		  CASE uiBothStep OF
           		0://	
					BoxReady_1st := FALSE;
					BoxReady_2nd := FALSE;					
					uiBothStep:=1000;	
	
				1000:
						BoxReady_1st:=TRUE;
						uiBothStep:=2000;
						
				2000:
						IF Robot._DI1.Notification THEN
							uiBothStep:=3000;
						END_IF
				3000:
					
					
						uiBothStep:=9000;	
					
				9000:
						BoxReady_2nd:=TRUE;
						uiBothStep:=9999;
				
				9999: //Wait		
        // wait reset
        END_CASE

       	  // Robot Abs move
           		 Robot.M_StartRobotAbsMove( GetBox:=Get,
											UseClampA:=UseA,
											UseClampB:=UseB,
											Area:=Area,
											ClampA_Address:=Address_A,
											ClampB_Address:=Address_B,
											BoxReady_1:=BoxReady_1st,
											BoxReady_2:=BoxReady_2nd);	
		
		
        IF Robot._DI1.Done THEN
			tonTimeOut.IN:=FALSE;
            uiExecutingStep := 30080;
        END_IF
		IF tonTimeOut.Q=TRUE THEN
				tonTimeOut.IN:=FALSE;
				strStatus :='FB_ShippingRobot_Left Step 30000: Reset Robot timeout';
				_Error:=TRUE;
			END_IF
    30080: // Check robot command is clear
        
        Robot.M_ResetRobotAbsMove(UseA,UseB);

        IF NOT Robot._DI1.Done THEN
			tonTimeOut.IN:=FALSE;
            uiExecutingStep := 90000; // go to place step
        END_IF    
   		tonTimeOut.IN:=TRUE;
		IF tonTimeOut.Q=TRUE THEN
			strStatus :='FB_ShippingRobot_Left Step 30080: Stop Robot timeout';
			_Error:=TRUE;
		END_IF
		
	90000:
			IF bCompleteRequest THEN
				uiExecutingStep := 91000;
			ELSE
				uiExecutingStep := 99000;
			END_IF
			
	91000:	// shipping allocate mission complete signal
		BuzzBlinker(ENABLE:=TRUE , TIMELOW:=T#0.3S , TIMEHIGH:=T#0.3S , OUT=> Buzz);
		LightBlinker(ENABLE := TRUE , TIMELOW := T#0.3S , TIMEHIGH := T#0.3S , OUT => RedLamp );
		TrigBuzz(CLK:=Buzz);
		TrigLight(CLK :=RedLamp);
		IF TrigBuzz.Q THEN
			BlinkInfo.BuzzCount := BlinkInfo.BuzzCount +1;
		END_IF
		IF TrigLight.Q THEN
			BlinkInfo.LightCount := BlinkInfo.LightCount +1;
		END_IF
		
		IF BlinkInfo.BuzzCount >= BlinkInfo.MaxBuzzCOunt AND BlinkInfo.LightCount >=BlinkInfo.MaxLightCount THEN
			TON_BlinkDelay.IN :=TRUE;
			IF TON_BlinkDelay.q THEN
				uiExecutingStep := 99000;
			END_IF
		END_IF
   
    99000: // process done
		TON_BlinkDelay.IN := FALSE;
        Status    := 'FB_ShippingRobot_Left Step 99000: Process completed';
        _Executed := TRUE;
END_CASE

IF _Executed THEN
    eState := STATE_DONE;
ELSIF _Error THEN
	//FUN_UniqueErrorCodeGenerator(iErrorID := ErrorID,UinqueErrorCode=>_UniqueErrorCode);
    eState := STATE_ERROR;
ELSIF NOT Execute THEN
    eState := STATE_RESETTING;
END_IF
IF _Abort OR Abort THEN
	//FUN_UniqueErrorCodeGenerator(iErrorID := ErrorID,UinqueErrorCode=>_UniqueErrorCode);
	eSTATE:=STATE_ABORTING;
END_IF
END_METHOD

METHOD  M_STATE_RESETTING
VAR_INPUT
END_VAR
// Done := false 更改到Dormant 清除確保，上位檢查到done 後可以直接下Execute

CASE uiResettingStep OF

	0:
		bCompleteRequest := false;
		tonTimeOut.IN:=FALSE;
		TON_BlinkDelay.IN := FALSE;

		uiResettingStep := 100;

	100:
		Robot.M_ResetAllCommand();
		IF Robot.M_CheckResetAllCommand() THEN
			uiResettingStep := 9999;
		END_IF

	9999:
//		Done := FALSE;
//		Busy := FALSE;
		_ResetCompleted:=TRUE;
END_CASE

IF _ResetCompleted THEN
	eSTATE:=STATE_DORMANT;
END_IF
END_METHOD

END_FUNCTION_BLOCK

// ---- Library/20_MachineUnits/23_ShippingArea/RobotService/FB_ShippingRobot_Right.TcPOU
FUNCTION_BLOCK FB_ShippingRobot_Right EXTENDS FB_RobotRegionMove_BufferArea
VAR_INPUT
	Buzz	: REFERENCE TO BOOL;
	RedLamp	: REFERENCE TO BOOL;
	bCompleteRequest	: BOOL;
	Input		: REFERENCE TO ST_InputTable;
END_VAR
VAR_OUTPUT
	bTransCVInPosition : BOOL;
END_VAR
VAR
	//Area : E_RobotArea := E_RobotArea.TransmitCV_End;
	Blink		: ST_BlinkInfo;
	BuzzBlinker	: Blink;
	LightBlinker: Blink;
	TrigBuzz	: R_TRIG;
	TrigLight	: R_TRIG;
	BlinkInfo	: ST_BlinkInfo;
	
	TON_BlinkDelay	: TON;
END_VAR

SUPER^.A10_StateControl();
A00_BasicUnits();
Area := E_RobotArea.ShippingRobotRight;

ACTION A00_BasicUnits:
tonTimeOut(PT:=T#60S);
TON_BlinkDelay(PT:= T#1S);

bTransCVInPosition := Input.bShippingTransCV_Rightside_Arrived;
ErrorID:=2250;
END_ACTION

METHOD M_CheckCommand : BOOL // True : Command is useful
VAR_INPUT
END_VAR
VAR
	
END_VAR
// Check command paremeter is correct

THIS^.Get :=Info.Get;
UseA := Info.UseA;
UseB := Info.UseB;
//Buffer area
		
IF UseA AND ( Info.A_Position<1 OR  Info.A_Position>40) THEN
	strStatus:='FB_ShippingRobot_Right: Wrong command ,Position A Not allow';
	M_CheckCommand:=FALSE;
	RETURN;			
END_IF		

IF UseB AND( Info.B_Position<1 OR  Info.B_Position>40 )THEN
	strStatus:='FB_ShippingRobot_Right: Wrong command ,Position B Not allow';
	M_CheckCommand:=FALSE;
	RETURN;			
END_IF
		
IF Get THEN
	IF NOT Robot._DI1.ClampA_Open THEN
		strStatus := 'FB_ShippingRobot_Right: Get command , clamp have box ';
		M_CheckCommand := FALSE;
		RETURN;
	END_IF
ELSE
	IF Robot._DI1.ClampA_Open THEN 
		strStatus := 'FB_ShippingRobot_Right: Place command , clamp not have box ';
		M_CheckCommand := FALSE;
		RETURN;
	END_IF
END_IF
M_CheckCommand:=TRUE;
END_METHOD

METHOD M_CheckUnitsNotBusy : BOOL
VAR_INPUT
END_VAR
M_CheckUnitsNotBusy := true;
END_METHOD

METHOD M_CheckUnitsReady : BOOL
VAR_INPUT
END_VAR
M_CheckUnitsReady := true;
END_METHOD

METHOD  M_STATE_ABORTED
VAR_INPUT
END_VAR
ERROR :=TRUE;
Busy    := FALSE;
Aborted := TRUE;
Status := strStatus;
_AbortCompleted := FALSE;
uiAbortingStep := 0;
UniqueErrorCode:=_UniqueErrorCode;

IF NOT Execute THEN
	eSTATE:=STATE_RESETTING;
END_IF

IF Execute AND Reset THEN
		Error := FALSE;
	Aborted := false;
	uiExecutingStep :=uiResumeStep;
	PreviousStrStatus := strStatus;
	PreviousErrorCode := _UniqueErrorCode;

	eSTATE:=STATE_EXECUTING;
END_IF
END_METHOD

METHOD  M_STATE_ABORTING
VAR_INPUT
END_VAR
CASE uiAbortingStep OF
	0 :
		_Abort := FALSE;
		Abort 			:= false;
		uiAbortingStep:=9999;
		tonTimeOut.IN := FALSE;
		IF strStatus = PreviousStrStatus THEN
			_UniqueErrorCode :=PreviousErrorCode;
		END_IF
		_Abort :=FALSE;
	9999:	_AbortCompleted:=TRUE;
END_CASE

IF _AbortCompleted THEN	
	eSTATE :=STATE_ABORTED;
END_IF
END_METHOD

METHOD  M_STATE_DONE
VAR_INPUT
END_VAR
Busy   := FALSE;
_Error := Error := FALSE;
_Abort := Abort := FALSE;
Done   := TRUE;

IF NOT Execute THEN
    eState := STATE_RESETTING;
END_IF
END_METHOD

METHOD  M_STATE_DORMANT
VAR_INPUT
END_VAR
// Clear FB output
Busy            := FALSE;
Done            := FALSE;
Aborted         := FALSE;
Error           := FALSE;
ErrorID         := 0;
Status          := '';
_ResetCompleted := FALSE;
_Error          := FALSE;
_Executed       := FALSE;

bCompleteRequest := false;
TON_BlinkDelay.IN := FALSE;
tonTimeOut.IN:=FALSE;
strStatus :='FB_ShippingRobot_Right: No Error';
uiExecutingStep :=uiResettingStep :=uiResumeStep :=0;
PreviousStrStatus			 :='';
PreviousErrorCode			 :='';
_UniqueErrorCode	:='0';

// Wait Execute command
IF Execute AND bTransCVInPosition THEN
    eState := STATE_EXECUTING;
ELSE
	strStatus :='FB_ShippingRobot_Right: Wrong command ,TransCV not In Position ';
	_ERROR := TRUE;
END_IF
END_METHOD

METHOD  M_STATE_ERROR
VAR_INPUT
END_VAR
ERROR   :=TRUE;
Busy	:=FALSE;
Status := strStatus;
UniqueErrorCode:=_UniqueErrorCode;
IF NOT Execute THEN	
eSTATE:=STATE_RESETTING;
END_IF
END_METHOD

METHOD  M_STATE_EXECUTING
VAR_INPUT
END_VAR
VAR_INST
    ActionMode       : E_ReloadRoundBoxAction;
	BoxReady_1st : BOOL;
	BoxReady_2nd : BOOL;
    CarrierReady_1st : BOOL;
    CarrierReady_2nd : BOOL;
    uiBothStep : UINT;
    uiSingleClampStep : UINT;
	Address_A : INT;
	Address_B : INT;
END_VAR
VAR
	WareHouse: INT;
END_VAR
// Set Busy active edit by johnson
Busy := TRUE;
IF THIS^.Stop THEN // Pending the timeout when Stop signal occur
	tonTimeout.IN :=FALSE;
END_IF
// Service Process
CASE uiExecutingStep OF
	0:
        // Clear variable
        ActionMode       := E_ReloadRoundBoxAction.Undefined;
        CarrierReady_1st := FALSE;
        CarrierReady_2nd := FALSE;
        uiBothStep := 0;
		uiSingleClampStep :=0;
		BoxReady_1st := 0;
		BoxReady_2nd := 0;
		tonTimeOut.IN:=FALSE;
        // Check command
        IF M_CheckCommand() THEN
            uiExecutingStep := 10;
		ELSE
			_Error:=TRUE;
        END_IF
    10:
        // Start process, check units first
        IF M_CheckUnitsReady() THEN
            uiExecutingStep := 20;
        END_IF
    20:
        // CHeck units not busy state
        IF M_CheckUnitsNotBusy() THEN
            uiExecutingStep := 1000;
        END_IF
   
	1000:   
			// Read   coordinate
 			 Address_A := LREAL_TO_INT(Info.A_Position);
			 Address_B := LREAL_TO_INT(Info.B_Position);
			 
			IF UseA AND NOT UseB THEN
				//Only clampA
				uiExecutingStep := 10000;
			ELSIF NOT UseA AND UseB THEN
				//Only ClampB 
				uiExecutingStep := 20000;
			ELSIF UseA AND UseB THEN
				//Both Clamps
				uiExecutingStep := 30000;		
			END_IF
       
    10000: // Only ClampA 
        IF NOT Robot._DI1.Done THEN            
           		BoxReady_1st:=TRUE;				
			          		 
				  // Robot Abs move
           		 Robot.M_StartRobotAbsMove(GetBox:=Get,
											UseClampA:=UseA,
											UseClampB:=UseB,
											Area:=Area,
											ClampA_Address:=Address_A,
											ClampB_Address:=Address_B,
											BoxReady_1:=BoxReady_1st,
											BoxReady_2:=BoxReady_2nd);	  
		
        ELSE
			tonTimeOut.IN:=FALSE;
            uiExecutingStep := 10080;
        END_IF
		tonTimeOut.IN:=TRUE;
		IF tonTimeOut.Q=TRUE THEN
			tonTimeOut.IN:=FALSE;			
			strStatus :='FB_ShippingRobot_Right Step 10000: Action Robot timeout';
			_Abort:=TRUE;
			uiResettingStep := 10000;
		END_IF	
		IF Robot.Error THEN
			_Abort := TRUE;
			strStatus := 'FB_ShippingRobot_Right Step 10000: FB_ShippingRobot place box to right Plate , Robot Error';
			uiResettingStep := 10000;
		END_IF
		
    10080:
        Robot.M_ResetRobotAbsMove(UseA,UseB); // Clear command and go to place box
		tonTimeOut.IN:=TRUE;
        IF NOT Robot._DI1.Done THEN
			tonTimeOut.IN:=FALSE;
            uiExecutingStep := 90000; 
        END_IF
    	IF tonTimeOut.Q=TRUE THEN
			strStatus :='FB_ShippingRobot_Right Step 10080: Reset Robot timeout';
			uiResettingStep := 10080;
			_Abort:=TRUE;
		END_IF
    
   20000: // Only ClampB
        IF NOT Robot._DI1.Done THEN           		
				BoxReady_2nd:=TRUE;				          		 
				  // Robot Abs move
           		 Robot.M_StartRobotAbsMove( GetBox:=Get,
											UseClampA:=UseA,
											UseClampB:=UseB,
											Area:=Area,
											ClampA_Address:=Address_A,
											ClampB_Address:=Address_B,
											BoxReady_1:=BoxReady_1st,
											BoxReady_2:=BoxReady_2nd);	
        ELSE
			tonTimeOut.IN:=FALSE;
            uiExecutingStep := 20080;
        END_IF
		tonTimeOut.IN:=TRUE;
			IF tonTimeOut.Q=TRUE THEN
				tonTimeOut.IN:=FALSE;
				strStatus :='FB_ShippingRobot_Right Step 20000: Reset Robot timeout';
				_Error:=TRUE;
			END_IF
    20080:
       Robot.M_ResetRobotAbsMove(UseA,UseB);; // Clear command 

        IF NOT Robot._DI1.Done THEN
            uiExecutingStep := 90000; 
        END_IF
		tonTimeOut.IN:=TRUE;
		IF tonTimeOut.Q=TRUE THEN
			strStatus :='FB_ShippingRobot_Right Step 20080: Reset Robot timeout';
			_Error:=TRUE;
		END_IF
    30000: // Both Clamps
        		
		
		  CASE uiBothStep OF
           		0://	
					BoxReady_1st := FALSE;
					BoxReady_2nd := FALSE;					
					uiBothStep:=1000;	
	
				1000:
						BoxReady_1st:=TRUE;
						uiBothStep:=2000;
						
				2000:
						IF Robot._DI1.Notification THEN
							uiBothStep:=3000;
						END_IF
				3000:
					
					
						uiBothStep:=9000;	
					
				9000:
						BoxReady_2nd:=TRUE;
						uiBothStep:=9999;
				
				9999: //Wait		
        // wait reset
        END_CASE

       	  // Robot Abs move
           		 Robot.M_StartRobotAbsMove( GetBox:=Get,
											UseClampA:=UseA,
											UseClampB:=UseB,
											Area:=Area,
											ClampA_Address:=Address_A,
											ClampB_Address:=Address_B,
											BoxReady_1:=BoxReady_1st,
											BoxReady_2:=BoxReady_2nd);	
		
		
        IF Robot._DI1.Done THEN
			tonTimeOut.IN:=FALSE;
            uiExecutingStep := 30080;
        END_IF
		IF tonTimeOut.Q=TRUE THEN
				tonTimeOut.IN:=FALSE;
				strStatus :='FB_ShippingRobot_Right Step 30000: Reset Robot timeout';
				_Error:=TRUE;
			END_IF
    30080: // Check robot command is clear
        
        Robot.M_ResetRobotAbsMove(UseA,UseB);

        IF NOT Robot._DI1.Done THEN
			tonTimeOut.IN:=FALSE;
            uiExecutingStep := 90000; // go to place step
        END_IF    
   		tonTimeOut.IN:=TRUE;
		IF tonTimeOut.Q=TRUE THEN
			strStatus :='FB_ShippingRobot_Right Step 30080: Stop Robot timeout';
			_Error:=TRUE;
		END_IF
   
	90000:
			IF bCompleteRequest THEN
				uiExecutingStep := 91000;
			ELSE
				uiExecutingStep := 99000;
			END_IF
			
	91000:	// shipping allocate mission complete signal
		BuzzBlinker(ENABLE:=TRUE , TIMELOW:=T#0.3S , TIMEHIGH:=T#0.3S , OUT=> Buzz);
		LightBlinker(ENABLE := TRUE , TIMELOW := T#0.3S , TIMEHIGH := T#0.3S , OUT => RedLamp );
		TrigBuzz(CLK:=Buzz);
		TrigLight(CLK :=RedLamp);
		IF TrigBuzz.Q THEN
			BlinkInfo.BuzzCount := BlinkInfo.BuzzCount +1;
		END_IF
		IF TrigLight.Q THEN
			BlinkInfo.LightCount := BlinkInfo.LightCount +1;
		END_IF
		
		IF BlinkInfo.BuzzCount >= BlinkInfo.MaxBuzzCOunt AND BlinkInfo.LightCount >=BlinkInfo.MaxLightCount THEN
			TON_BlinkDelay.IN :=TRUE;
			IF TON_BlinkDelay.q THEN
				uiExecutingStep := 99000;
			END_IF
		END_IF
   
		
    99000: // process done
		TON_BlinkDelay.IN := FALSE;
        Status    := 'FB_ShippingRobot_Right Step 99000: Process completed';
        _Executed := TRUE;
END_CASE

IF _Executed THEN
    eState := STATE_DONE;
ELSIF _Error THEN
	//FUN_UniqueErrorCodeGenerator(iErrorID := ErrorID,UinqueErrorCode=>_UniqueErrorCode);
    eState := STATE_ERROR;
ELSIF NOT Execute THEN
    eState := STATE_RESETTING;
END_IF
IF _Abort OR Abort THEN
	//FUN_UniqueErrorCodeGenerator(iErrorID := ErrorID,UinqueErrorCode=>_UniqueErrorCode);
	eSTATE:=STATE_ABORTING;
END_IF
END_METHOD

METHOD  M_STATE_RESETTING
VAR_INPUT
END_VAR
Busy := TRUE;
Error := FALSE;


CASE uiResettingStep OF

	0:
		bCompleteRequest := false;
		TON_BlinkDelay.IN := FALSE;
		tonTimeOut.IN:=FALSE;
		//Robot.M_ResetAllCommand();
		Robot.M_ResetRobotAbsMove(TRUE,TRUE);

		uiResettingStep:=9999;
	9999:
		Done := FALSE;
		Busy := FALSE;
		_ResetCompleted:=TRUE;
END_CASE
IF _ResetCompleted THEN
	eSTATE:=STATE_DORMANT;
END_IF
END_METHOD

END_FUNCTION_BLOCK

// ---- Library/20_MachineUnits/23_ShippingArea/RobotService/FB_ShippingRobot_Buffer.TcPOU
FUNCTION_BLOCK FB_ShippingRobot_Buffer EXTENDS FB_RobotRegionMove_BufferArea
VAR_INPUT
	Input	: REFERENCE TO ST_InputTable;
	Output	: REFERENCE TO ST_OutputTable;
	Cylinder: REFERENCE TO UNI_CylinderList;
END_VAR
VAR_OUTPUT
END_VAR
VAR
	HasBufferArea		: BOOL:= FALSE;		// 直接在這裡切換True/False 就能判斷程式內部是否有判斷緩衝區機構了。>> false 無機構，True 有機構
	// 用於轉型 Lreal
	iCmdPosA	: INT;
	
	TON_RobotActionTimeOut		: TON;
	TON_CheckRobotDoneTimeOut	: TON;
	
	uiGetStep	: UDINT;
END_VAR

THIS^.A00_BasicUnits();
SUPER^.A10_StateControl();

Area := E_RobotArea.ShippingBufferArea;

ACTION A00_BasicUnits:
TON_RobotActionTimeOut( PT := T#60S);
TON_CheckRobotDoneTimeOut(PT := T#30S);
END_ACTION

METHOD M_CheckCommandVaild : BOOL
VAR_INPUT
END_VAR
VAR
END_VAR
THIS^.Get :=Info.Get;
UseA := Info.UseA;
UseB := Info.UseB;

// 出貨區小手臂只有 A爪,所以程式內只有判斷 useA
IF UseB THEN
	M_CheckCommandVaild := FALSE;
	status 				:= 'FB_ShippingRobot_Buffer: not have B Clamp , not can retry';
	RETURN;
END_IF
IF NOT UseA THEN
	M_CheckCommandVaild := FALSE;
	status 				:= 'FB_ShippingRobot_Buffer: A Clamp must be used';
	RETURN;
END_IF

// 預防上位給予的位置是小數點
IF info.A_Position <> INT_TO_LREAL(LREAL_TO_INT(info.A_Position)) THEN
	M_CheckCommandVaild := FALSE;
	status 				:= 'FB_ShippingRobot_Buffer: A_Position not integer ,not can retry';
	RETURN;
END_IF

iCmdPosA := LREAL_TO_INT(info.A_Position);

IF NOT ((iCmdPosA >= 1) AND (iCmdPosA <= 55))  THEN
	M_CheckCommandVaild := FALSE;
	status 				:= 'FB_ShippingRobot_Buffer: Position not valid ,not can retry';
	RETURN;
END_IF


IF Get THEN
	IF NOT Robot._DI1.ClampA_Open THEN
		status 				:= 'FB_ShippingRobot_Buffer: Get command , clamp have box ';
		M_CheckCommandVaild := FALSE;
		RETURN;
	END_IF
ELSE
	IF Robot._DI1.ClampA_Open THEN 
		status 				:= 'FB_ShippingRobot_Buffer: Place command , clamp not have box ';
		M_CheckCommandVaild := FALSE;
		RETURN;
	END_IF
END_IF

M_CheckCommandVaild := TRUE;
END_METHOD

METHOD  M_STATE_ABORTED
VAR_INPUT
END_VAR
Busy  := FALSE;
Error := TRUE;
Aborted := TRUE;
uiAbortingStep 	:= 0;
_AbortCompleted := FALSE;

// 狀態機切換
IF NOT Execute THEN
	eState := STATE_RESETTING;
ELSIF Execute AND reset THEN
	Error	:= false;
	Aborted	:= false;
	eState 	:= STATE_EXECUTING;
END_IF
END_METHOD

METHOD  M_STATE_ABORTING
VAR_INPUT
END_VAR
CASE uiAbortingStep OF
	0 :
		_Abort := FALSE;
		TON_RobotActionTimeOut.IN 	 := FALSE;
		TON_CheckRobotDoneTimeOut.IN := FALSE;
		
		uiAbortingStep:=9999;

	9999:	
		_AbortCompleted:=TRUE;
END_CASE

IF _AbortCompleted THEN	
	eSTATE :=STATE_ABORTED;
END_IF
END_METHOD

METHOD  M_STATE_DONE
VAR_INPUT
END_VAR
Busy   := FALSE;
_Error := Error := FALSE;
_Abort := Abort := FALSE;
Done   := TRUE;

IF NOT Execute THEN
    eState := STATE_RESETTING;
END_IF
END_METHOD

METHOD  M_STATE_DORMANT
VAR_INPUT
END_VAR
Busy 			:= FALSE;
Done 			:= FALSE;
Aborted 		:= FALSE;
Error			:= FALSE;
Paused			:= FALSE;
ErrorID			:= 0;
Status			:= '';
UniqueErrorCode := '';

_Executed 			:= FALSE;
_Error				:= FALSE;
_Abort				:= FALSE;
_ResetCompleted 	:= FALSE;
_AbortCompleted 	:= FALSE;
_HoldingCompleted 	:= FALSE;
_HeldCompleted	 	:= FALSE;
_UnholdCompleted 	:= FALSE;

uiExecutingStep 	:= 0;
uiResettingStep 	:= 0;
uiAbortingStep 		:= 0;
uiHoldingStep		:= 0;
uiHeldStep			:= 0;
uiUnholdStep		:= 0;
uiGetStep			:= 0;

TON_RobotActionTimeOut.IN 	 := FALSE;
TON_CheckRobotDoneTimeOut.IN := FALSE;

IF Execute AND HasBufferArea THEN
    eState := STATE_EXECUTING;
ELSIF  Execute AND NOT HasBufferArea THEN
	Status := 'FB_ShippingRobot_Buffer: Wrong Comman Not have bufferArea in ShippingArea';
	eState := STATE_ERROR;
END_IF
END_METHOD

METHOD  M_STATE_ERROR
VAR_INPUT
END_VAR
ERROR   := TRUE;
Busy	:= FALSE;
_Error	:= false;

IF NOT Execute THEN	
	Error	:= FALSE;
	eSTATE	:=STATE_RESETTING;
END_IF
END_METHOD

METHOD  M_STATE_EXECUTING
VAR_INPUT
END_VAR
VAR_INST
	Address_A	 : INT;
	BoxReady_1st : BOOL;
END_VAR
busy := true;

// 暫停
IF Pause THEN 
	_HoldingCompleted 	:= FALSE;
	_HeldCompleted	 	:= FALSE;
	_UnholdCompleted 	:= FALSE;
	uiHoldingStep		:= 0;
	uiHeldStep			:= 0;
	uiUnholdStep		:= 0;
	eState    			:= STATE_Holding;
END_IF

// 動作主流程 狀態機
CASE uiExecutingStep OF
	
	0:		// init 
			BoxReady_1st := FALSE;		
			Address_A	 := 0;
			
			uiExecutingStep := 100;
		
	100:	// 檢查命令是否是有效值
			IF M_CheckCommandVaild() THEN
				uiExecutingStep := 1000;
			ELSE
				_Error := TRUE;
			END_IF
			
	1000:	// 注入位置座標
			Address_A 		:= iCmdPosA;
			uiExecutingStep := 10000;
			
	10000:	// RobotAction
			TON_RobotActionTimeOut.IN := TRUE;
			IF NOT Robot._DI1.Done THEN  
				IF Get THEN
					// 取盒動作先判斷盒子的目標位置，去選擇接下來的動作。
					CASE uiGetStep OF
							0:	
								CASE Address_A OF
									1..54:
											uiGetStep := 400;
									55:
											uiGetStep := 100;
								END_CASE
								
							100:
								Cylinder.List.fbShippingBuffer_Press.M_Extend();
								IF Cylinder.List.fbShippingBuffer_Press.InFrontPosition THEN
									uiGetStep := 300;
								END_IF						
							300:
								Cylinder.List.fbShippingBuffer_Press.M_Retract();
								IF Cylinder.List.fbShippingBuffer_Press.InRearPosition THEN
									uiGetStep := 400;
								END_IF
							400:
								BoxReady_1st := TRUE;
						END_CASE
						
					 Robot.M_StartRobotAbsMove(GetBox:=TRUE,
												UseClampA:=UseA,
												UseClampB:=FALSE,
												Area:=Area,
												ClampA_Address:=Address_A,
												ClampB_Address:=0,
												BoxReady_1:=BoxReady_1st,
												BoxReady_2:=FALSE);	  
				
				ELSE
					
					IF Cylinder.List.fbShippingBuffer_Press.InRearPosition THEN
						BoxReady_1st:=TRUE;
					ELSE
						Cylinder.List.fbShippingBuffer_Press.M_Retract();
					END_IF
					
					Robot.M_StartRobotAbsMove(GetBox:=FALSE,
												UseClampA:=UseA,
												UseClampB:=FALSE,
												Area:=Area,
												ClampA_Address:=Address_A,
												ClampB_Address:=0,
												BoxReady_1:=BoxReady_1st,
												BoxReady_2:=FALSE);	
				END_IF
			ELSE
				uiExecutingStep := 11000;
			END_IF
			
			IF TON_RobotActionTimeOut.Q  THEN
				_Abort 	:= TRUE;
				Status	:= 'FB_ShippingRobot_Buffer Step 10000: RobotAction Timeout,can retry';
			END_IF
			IF Robot.Error THEN
				Status := CONCAT('FB_ShippingRobot place Left Plate Error',robot.ErrMsg);
				_Abort := TRUE;
		END_IF
			
	11000:	// reset 手臂命令
			Robot.M_ResetRobotAbsMove(UseA,UseB); // Clear command and go to place box
			TON_RobotActionTimeOut.IN 	 := FALSE;
			TON_CheckRobotDoneTimeOut.IN := TRUE;
			IF NOT Robot._DI1.Done THEN
				TON_CheckRobotDoneTimeOut.IN := FALSE;
            	uiExecutingStep := 90000; 
        	END_IF
			IF TON_CheckRobotDoneTimeOut.Q THEN
				_Error := TRUE;
				status := 'FB_ShippingRobot_Buffer Step 11000: Wait Robot done Timeout';
			END_IF

	90000:
			TON_CheckRobotDoneTimeOut.IN := FALSE;
			Status    := 'FB_ShippingRobot_Buffer Step 90000: Process completed';
        	_Executed := TRUE;
end_case

// 狀態機切換
IF NOT Execute THEN
	eState := STATE_RESETTING;
ELSIF _Error THEN
	eState := STATE_ERROR;
ELSIF _Abort THEN
	eState := STATE_ABORTING;
ELSIF _Executed THEN
	eState := STATE_DONE;
END_IF
END_METHOD

METHOD M_STATE_HELD
VAR_INPUT
END_VAR

Busy 	:= FALSE;
Paused 	:= TRUE;

CASE uiHeldStep OF
	0:
		uiHeldStep := 9999;

	9999:
		_HeldCompleted := TRUE;	

END_CASE

IF _HeldCompleted AND NOT Pause THEN
	eState := STATE_UnHold;
END_IF
END_METHOD

METHOD M_STATE_HOLDING
VAR_INPUT
END_VAR

CASE uiHoldingStep OF 
	0:	    // 需關閉 Timer 等等須暫停的變數
		TON_RobotActionTimeOut.IN 	 := FALSE;
		TON_CheckRobotDoneTimeOut.IN := FALSE;
		
		uiHoldingStep := 9999;
		
	9999:	// holding 完成
		_HoldingCompleted := TRUE;
END_CASE

IF _HoldingCompleted THEN
	eState := STATE_Held;
END_IF
END_METHOD

METHOD  M_STATE_RESETTING
VAR_INPUT
END_VAR
// Done := false 更改到Dormant 清除確保，上位檢查到done 後可以直接下Execute

CASE uiResettingStep OF

	0:
		IF Cylinder.List.fbShippingBuffer_Press.InRearPosition THEN
			uiResettingStep := 100;
		ELSE
			Cylinder.List.fbShippingBuffer_Press.M_Retract();
		END_IF

	100:
		Robot.M_ResetAllCommand();
		IF Robot.M_CheckResetAllCommand() THEN
			uiResettingStep := 9999;
		END_IF

	9999:
//		Done := FALSE;
//		Busy := FALSE;
		_ResetCompleted:=TRUE;

END_CASE

IF _ResetCompleted THEN
	eSTATE:=STATE_DORMANT;
END_IF
END_METHOD

METHOD M_STATE_UNHOLD
VAR_INPUT
END_VAR
CASE uiUnholdStep OF 
	0:		
		uiUnholdStep := 9999;
		
	9999:
		_UnholdCompleted := TRUE;
		
END_CASE

IF _UnholdCompleted THEN
	Paused := FALSE;
	eState := STATE_EXECUTING;
END_IF
END_METHOD

END_FUNCTION_BLOCK

// ---- Library/20_MachineUnits/23_ShippingArea/RobotService/FB_ShippingRobot_PhotoStandByPos.TcPOU
FUNCTION_BLOCK FB_ShippingRobot_PhotoStandByPos EXTENDS FB_RobotRegionMove_BufferArea
VAR_INPUT
	Input	: REFERENCE TO ST_InputTable;
	Output	: REFERENCE TO ST_OutputTable;
END_VAR
VAR_OUTPUT
END_VAR
VAR
	// 用於轉型 Lreal
	iCmdPosA	: INT;
	
	TON_RobotActionTimeOut		: TON;
	TON_CheckRobotDoneTimeOut	: TON;
	
END_VAR

THIS^.A00_BasicUnits();
SUPER^.A10_StateControl();

Area := E_RobotArea.ShippingCCDPos;

ACTION A00_BasicUnits:
TON_RobotActionTimeOut( PT := T#60S);
TON_CheckRobotDoneTimeOut(PT := T#30S);
END_ACTION

METHOD M_CheckCommandVaild : BOOL
VAR_INPUT
END_VAR
VAR
END_VAR
THIS^.Get :=Info.Get;
UseA := Info.UseA;
UseB := Info.UseB;

// 出貨區小手臂只有 A爪,所以程式內只有判斷 useA
IF UseB THEN
	M_CheckCommandVaild := FALSE;
	status 				:= 'FB_ShippingRobot_PhotoStandByPos: WrongCommand not have B Clamp , not can retry';
	RETURN;
END_IF
IF NOT UseA THEN
	M_CheckCommandVaild := FALSE;
	status 				:= 'FB_ShippingRobot_PhotoStandByPos: WrongCommand A Clamp must be used';
	RETURN;
END_IF

//
IF info.A_Position <> 0 THEN
	M_CheckCommandVaild := TRUE;
	status				:= 'FB_ShippingRobot_PhotoStandByPos: WrongCommand not have Position';
END_IF

M_CheckCommandVaild := TRUE;
END_METHOD

METHOD  M_STATE_ABORTED
VAR_INPUT
END_VAR

Busy  := FALSE;
Error := TRUE;
Aborted := TRUE;
uiAbortingStep 	:= 0;
_AbortCompleted := FALSE;

// 狀態機切換
IF NOT Execute THEN
	eState := STATE_RESETTING;
ELSIF Execute AND reset THEN
	Error	:= false;
	Aborted	:= false;
	eState 	:= STATE_EXECUTING;
END_IF
END_METHOD

METHOD  M_STATE_ABORTING
VAR_INPUT
END_VAR

CASE uiAbortingStep OF
	0 :
		_Abort := FALSE;
		TON_RobotActionTimeOut.IN 	 := FALSE;
		TON_CheckRobotDoneTimeOut.IN := FALSE;
		
		uiAbortingStep:=9999;

	9999:	
		_AbortCompleted:=TRUE;
END_CASE

IF _AbortCompleted THEN	
	eSTATE :=STATE_ABORTED;
END_IF
END_METHOD

METHOD  M_STATE_DONE
VAR_INPUT
END_VAR
Busy   := FALSE;
_Error := Error := FALSE;
_Abort := Abort := FALSE;
Done   := TRUE;

IF NOT Execute THEN
    eState := STATE_RESETTING;
END_IF
END_METHOD

METHOD  M_STATE_DORMANT
VAR_INPUT
END_VAR
Busy 			:= FALSE;
Done 			:= FALSE;
Aborted 		:= FALSE;
Error			:= FALSE;
Paused			:= FALSE;
ErrorID			:= 0;
Status			:= '';
UniqueErrorCode := '';

_Executed 			:= FALSE;
_Error				:= FALSE;
_Abort				:= FALSE;
_ResetCompleted 	:= FALSE;
_AbortCompleted 	:= FALSE;
_HoldingCompleted 	:= FALSE;
_HeldCompleted	 	:= FALSE;
_UnholdCompleted 	:= FALSE;

uiExecutingStep 		:= 0;
uiResettingStep 		:= 0;
uiAbortingStep 			:= 0;
uiHoldingStep			:= 0;
uiHeldStep				:= 0;
uiUnholdStep			:= 0;

TON_RobotActionTimeOut.IN 	 := FALSE;
TON_CheckRobotDoneTimeOut.IN := FALSE;

IF Execute THEN
    eState := STATE_EXECUTING;
END_IF
END_METHOD

METHOD  M_STATE_ERROR
VAR_INPUT
END_VAR

ERROR   := TRUE;
Busy	:= FALSE;
_Error	:= false;

IF NOT Execute THEN	
	Error	:= FALSE;
	eSTATE	:=STATE_RESETTING;
END_IF
END_METHOD

METHOD  M_STATE_EXECUTING
VAR_INPUT
END_VAR
VAR_INST
	Address_A	 : INT;
	BoxReady_1st : BOOL;
END_VAR
busy := true;

// 暫停
IF Pause THEN 
	_HoldingCompleted 	:= FALSE;
	_HeldCompleted	 	:= FALSE;
	_UnholdCompleted 	:= FALSE;
	uiHoldingStep		:= 0;
	uiHeldStep			:= 0;
	uiUnholdStep		:= 0;
	eState    			:= STATE_Holding;
END_IF

// 動作主流程 狀態機
CASE uiExecutingStep OF
	
	0:		// 檢查命令是否是有效值
			IF M_CheckCommandVaild() THEN
				uiExecutingStep := 1000;
			ELSE
				_Error := TRUE;
			END_IF
			
	1000:	
			uiExecutingStep := 10000;
			
	10000:	// RobotAction
			TON_RobotActionTimeOut.IN := TRUE;
			IF NOT Robot._DI1.Done THEN  
			
					 Robot.M_StartRobotAbsMove(GetBox:=TRUE,
												UseClampA:=UseA,
												UseClampB:=FALSE,
												Area:=Area,
												ClampA_Address:=0,
												ClampB_Address:=0,
												BoxReady_1:=BoxReady_1st,
												BoxReady_2:=FALSE);	  
				
			ELSE
				uiExecutingStep := 11000;
			END_IF
			
			IF TON_RobotActionTimeOut.Q THEN
				_Abort 	:= TRUE;
				Status	:= 'FB_ShippingRobot_PhotoStandByPos Step 10000: RobotAction Timeout,can retry';
			END_IF
			
	11000:	// reset 手臂命令
			Robot.M_ResetRobotAbsMove(UseA,UseB); // Clear command and go to place box
			TON_RobotActionTimeOut.IN 	 := FALSE;
			TON_CheckRobotDoneTimeOut.IN := TRUE;
			IF NOT Robot._DI1.Done THEN
				TON_CheckRobotDoneTimeOut.IN := FALSE;
            	uiExecutingStep := 90000; 
        	END_IF
			IF TON_CheckRobotDoneTimeOut.Q THEN
				_Error := TRUE;
				status := 'FB_ShippingRobot_PhotoStandByPos Step 11000: Wait Robot done Timeout';
			END_IF
		
	90000:
			Status    := 'FB_ShippingRobot_PhotoStandByPos Step 90000: Process completed';
        	_Executed := TRUE;
end_case

// 狀態機切換
IF NOT Execute THEN
	eState := STATE_RESETTING;
ELSIF _Error THEN
	eState := STATE_ERROR;
ELSIF _Abort THEN
	eState := STATE_ABORTING;
ELSIF _Executed THEN
	eState := STATE_DONE;
END_IF
END_METHOD

METHOD M_STATE_HELD
VAR_INPUT
END_VAR

Busy 	:= FALSE;
Paused 	:= TRUE;

CASE uiHeldStep OF
	0:
		uiHeldStep := 9999;

	9999:
		_HeldCompleted := TRUE;	

END_CASE

IF _HeldCompleted AND NOT Pause THEN
	eState := STATE_UnHold;
END_IF
END_METHOD

METHOD M_STATE_HOLDING
VAR_INPUT
END_VAR

CASE uiHoldingStep OF 
	0:	// 需關閉 Timer 等等須暫停的變數
		TON_RobotActionTimeOut.IN 	 := FALSE;
		TON_CheckRobotDoneTimeOut.IN := FALSE;
		
		uiHoldingStep := 9999;
		
	9999:	// holding 完成
		_HoldingCompleted := TRUE;
END_CASE

IF _HoldingCompleted THEN
	eState := STATE_Held;
END_IF
END_METHOD

METHOD  M_STATE_RESETTING
VAR_INPUT
END_VAR
// Done := false 更改到Dormant 清除確保，上位檢查到done 後可以直接下Execute

CASE uiResettingStep OF

	0:
		TON_RobotActionTimeOut.IN	:= FALSE;
		TON_CheckRobotDoneTimeOut.IN:= FALSE;
		uiResettingStep := 100;

	100:
		Robot.M_ResetAllCommand();
		IF Robot.M_CheckResetAllCommand() THEN
			uiResettingStep := 9999;
		END_IF

	9999:
//		Done := FALSE;
//		Busy := FALSE;
		_ResetCompleted:=TRUE;
END_CASE

IF _ResetCompleted THEN
	eSTATE:=STATE_DORMANT;
END_IF
END_METHOD

METHOD M_STATE_UNHOLD
VAR_INPUT
END_VAR
CASE uiUnholdStep OF 
	0:		
		uiUnholdStep := 9999;
		
	9999:
		_UnholdCompleted := TRUE;
		
END_CASE

IF _UnholdCompleted THEN
	Paused := FALSE;
	eState := STATE_EXECUTING;
END_IF
END_METHOD

END_FUNCTION_BLOCK

// ---- Library/20_MachineUnits/23_ShippingArea/RobotService/FB_ShippingPlateScan.TcPOU
FUNCTION_BLOCK FB_ShippingPlateScan EXTENDS FB_ObjectBase_V2
VAR_INPUT
	Robot			: REFERENCE TO FB_FanucRobot_Basic_V2;
	Motor			: REFERENCE TO UNI_MotorList;			// 同尺寸軌道馬達 (Phase 2:只讀 InBackWard 狀態,不直接驅動)
	Cylinder		: REFERENCE TO UNI_CylinderList;		// Press1 / Press3 一次性伸出用
	SameSizeCVRequest	: REFERENCE TO ST_SameSizeCVRequest;	// Phase 2 仲裁:寫 bScan_NeedBackward,由 FB_MachineControl.A20_ConveyorArbitration 仲裁
	SameSizeCV_Press1_AlreadyExtended : REFERENCE TO BOOL;	// 一次性 latch (Press1):FALSE = 還沒伸過,本 FB 伸出後置 TRUE;TRUE = 跳過避免重伸
	SameSizeCV_Press3_AlreadyExtended : REFERENCE TO BOOL;	// 一次性 latch (Press3):同上
	Input			: REFERENCE TO ST_InputTable;			// SameSizeCV BoxNearShipping sensor
	Side			: E_ShippingPlateSide;		// Left=0 / Right=1
	PlateIndex		: E_ShippingPlateIndex;		// Plate1..Plate4 (enum 值 = 手臂 Position)
	ReadComplete	: BOOL;						// 上位讀完 PlateHasBox 後回 TRUE
END_VAR
VAR_OUTPUT
	PlateHasBox		: BOOL;		// Robot._DI13.9 (bClampA1_Laser_DetectStatus)
	FeedBack		: BOOL;		// 做完待上位讀,等 ReadComplete (做完才給,不是掃完)
END_VAR
VAR
	Area						: E_RobotArea;
	Address_A					: INT;

	TON_RobotActionTimeOut		: TON;
	TON_CheckRobotDoneTimeOut	: TON;
	TON_ScanTimeOut				: TON;
	TON_MechTimeOut				: TON;		// 軌道機構動作 watchdog (30s)
	tonBoxArriveDelay			: TON;		// Put 階段等盒到位 debounce (1s)
	TON_RobotCommandDelay		: TON;		// 延遲清除手臂程式跳出命令，會互卡到手臂_DO3 Execute。

	// Resume / Retry framework (對齊 FB_ShippingRobotTransfer 續做 pattern)
	uiResumeStep				: UDINT;	// retry / 續做進入點
	_bRetry						: BOOL;		// STATE_ABORTED 收到 Reset 後置 TRUE,觸發 retry
	_bAbsMoveStarted			: BOOL;		// 真的呼叫過 M_StartRobotAbsMove 才置 TRUE,防 stale Done 造成 ghost completion (對齊 FB_ShippingRobotTransfer)
	strStatus					: STRING;
	_UniqueErrorCode			: STRING;
	PreviousStrStatus			: STRING;
	PreviousErrorCode			: STRING;

	// Error blinking (Reset 後閃爍 1 秒,避開瞬間錯誤閃爍)
	trigErrorReset				: R_TRIG;
	tonErrorResetDelay			: TON;
	bErrorBlinking				: BOOL;
END_VAR

A00_BasicUnits();
SUPER^.A10_StateControl();

ACTION A00_BasicUnits:
TON_RobotActionTimeOut(PT := T#60S);
TON_CheckRobotDoneTimeOut(PT := T#30S);
TON_ScanTimeOut(PT := T#30S);
TON_MechTimeOut(PT := T#30S);
tonBoxArriveDelay(PT := T#1S);
TON_RobotCommandDelay(PT:= T#0.5S);

// Phase 2:軌道驅動移到 FB_MachineControl.A20_ConveyorArbitration,本 FB 只寫 SameSizeCVRequest.bScan_NeedBackward。
END_ACTION

METHOD PRIVATE M_ResolveAddress : BOOL
VAR_INPUT
END_VAR
// Side → Area
CASE Side OF
	E_ShippingPlateSide.Left:
		Area := E_RobotArea.ShippingRobotLeft;
	E_ShippingPlateSide.Right:
		Area := E_RobotArea.ShippingRobotRight;
ELSE
	strStatus := 'FB_ShippingPlateScan: invalid Side enum, not can retry';
	M_ResolveAddress := FALSE;
	RETURN;
END_CASE

// PlateIndex → Address (enum value 1..4 直接 = Position)
CASE PlateIndex OF
	E_ShippingPlateIndex.Plate1: Address_A := 1;
	E_ShippingPlateIndex.Plate2: Address_A := 2;
	E_ShippingPlateIndex.Plate3: Address_A := 3;
	E_ShippingPlateIndex.Plate4: Address_A := 4;
ELSE
	strStatus := 'FB_ShippingPlateScan: invalid PlateIndex enum, not can retry';
	M_ResolveAddress := FALSE;
	RETURN;
END_CASE

// Get=TRUE 需要爪是開的 (否則手臂在抓時會撞)
IF NOT Robot._DI1.ClampA_Open THEN
	strStatus := 'FB_ShippingPlateScan: ClampA must be open for scan/get';
	M_ResolveAddress := FALSE;
	RETURN;
END_IF

M_ResolveAddress := TRUE;
END_METHOD

METHOD M_STATE_ABORTED
VAR_INPUT
END_VAR
IF NOT _bRetry THEN
	Busy    := FALSE;
	Error   := TRUE;
	Aborted := TRUE;
	uiAbortingStep  := 0;
	_AbortCompleted := FALSE;
END_IF

IF Reset THEN
	_bRetry := TRUE;
	Error   := FALSE;
	Aborted := FALSE;
END_IF

IF NOT Execute THEN
	eState := STATE_RESETTING;
ELSIF Execute AND _bRetry AND NOT Robot._DI1.Error THEN
	// 續做:從上次 uiResumeStep 標的失敗點接續
	uiExecutingStep   := uiResumeStep;
	PreviousStrStatus := strStatus;
	PreviousErrorCode := _UniqueErrorCode;
	Status            := 'FB_ShippingPlateScan: no error';
	_bRetry           := FALSE;
	_bAbsMoveStarted  := FALSE;	// retry 進 EXECUTING 前清掉,讓 step 3100 ELSIF stale-Done 防護生效
	eState            := STATE_EXECUTING;
END_IF
END_METHOD

METHOD M_STATE_ABORTING
VAR_INPUT
END_VAR
// 對齊 FB_ShippingRobotTransfer ABORTING:reset robot 命令 → 等 Done 降 → Robot Error Recovery 循環
CASE uiAbortingStep OF
	0:
		_Abort := FALSE;
		Abort  := FALSE;
		TON_RobotActionTimeOut.IN    := FALSE;
		TON_CheckRobotDoneTimeOut.IN := FALSE;
		TON_ScanTimeOut.IN           := FALSE;
		TON_MechTimeOut.IN           := FALSE;
		tonBoxArriveDelay.IN         := FALSE;
		TON_RobotCommandDelay.IN	 := FALSE;
		// 撤銷軌道請求 (arbiter 看到沒人 request 會自動停)
		IF __ISVALIDREF(SameSizeCVRequest) THEN
			SameSizeCVRequest.bScan_NeedBackward := FALSE;
		END_IF
		_bAbsMoveStarted := FALSE;
		// 中斷 robot AbsMove 命令,避免 abort 期間 robot 還在跑舊軌跡
		Robot.M_ResetRobotAbsMove(TRUE, FALSE);
		uiAbortingStep := 50;

	50:	// 等 robot 命令真的被 reset 掉 (Done 降) 再進入錯誤檢查
		TON_CheckRobotDoneTimeOut.IN := TRUE;
		IF NOT Robot._DI1.Done THEN
			TON_CheckRobotDoneTimeOut.IN := FALSE;
			uiAbortingStep := 100;
		ELSIF TON_CheckRobotDoneTimeOut.Q THEN
			// reset 超時也繼續,後續 step 100 會處理 Robot.Error 路徑
			TON_CheckRobotDoneTimeOut.IN := FALSE;
			uiAbortingStep := 100;
		END_IF

	100:	// 看 robot 自己是否在 Error 狀態,需 robot error recovery
		IF Robot._DI1.Error THEN
			uiAbortingStep := 200;
		ELSE
			uiAbortingStep := 9999;
		END_IF

	200:	// Robot Error Recovery:對 robot 下 Reset 命令
		IF DAS_CoreSys.MachineControl.M_ShippingRobotResetCmd() THEN
			uiAbortingStep := 300;
		END_IF

	300:	// 對 robot 下 Start 命令重啟 prog
		IF DAS_CoreSys.MachineControl.M_ShippingRobotStartCmd() THEN
			uiAbortingStep := 400;
		END_IF

	400:	// 確認 robot 已脫離 error,還有就再循環一次
		IF Robot._DI1.Error THEN
			uiAbortingStep := 200;
		ELSE
			uiAbortingStep := 9999;
		END_IF

	9999:
		_AbortCompleted := TRUE;
END_CASE

IF _AbortCompleted THEN
	eState := STATE_ABORTED;
END_IF
END_METHOD

METHOD M_STATE_DONE
VAR_INPUT
END_VAR
Busy   := FALSE;
_Error := Error := FALSE;
_Abort := Abort := FALSE;
Done   := TRUE;

// Phase 2:撤銷軌道請求 (arbiter 仲裁,本 FB 不直接停 motor — 其他 FB 還在 request 時不應被影響)
IF __ISVALIDREF(SameSizeCVRequest) THEN
	SameSizeCVRequest.bScan_NeedBackward := FALSE;
END_IF

IF NOT Execute THEN
	eState := STATE_RESETTING;
END_IF
END_METHOD

METHOD M_STATE_DORMANT
VAR_INPUT
END_VAR
Busy            := FALSE;
Done            := FALSE;
Aborted         := FALSE;
Error           := FALSE;
Paused          := FALSE;
ErrorID         := 0;
Status          := '';
UniqueErrorCode := '';

_Executed         := FALSE;
_Error            := FALSE;
_Abort            := FALSE;
_ResetCompleted   := FALSE;
_AbortCompleted   := FALSE;
_HoldingCompleted := FALSE;
_HeldCompleted    := FALSE;
_UnholdCompleted  := FALSE;
_bRetry           := FALSE;
_bAbsMoveStarted  := FALSE;

uiExecutingStep := 0;
uiResettingStep := 0;
uiAbortingStep  := 0;
uiHoldingStep   := 0;
uiHeldStep      := 0;
uiUnholdStep    := 0;
uiResumeStep    := 0;

TON_RobotActionTimeOut.IN    := FALSE;
TON_CheckRobotDoneTimeOut.IN := FALSE;
TON_ScanTimeOut.IN           := FALSE;
TON_MechTimeOut.IN           := FALSE;
tonBoxArriveDelay.IN         := FALSE;
TON_RobotCommandDelay.IN	 := FALSE;

// Phase 2:撤銷軌道請求
IF __ISVALIDREF(SameSizeCVRequest) THEN
	SameSizeCVRequest.bScan_NeedBackward := FALSE;
END_IF

PlateHasBox := FALSE;
FeedBack    := FALSE;

PreviousStrStatus := '';
PreviousErrorCode := '';
_UniqueErrorCode  := '0';
bErrorBlinking    := FALSE;
tonErrorResetDelay.IN := FALSE;

IF Execute THEN
	eState := STATE_EXECUTING;
END_IF
END_METHOD

METHOD M_STATE_ERROR
VAR_INPUT
END_VAR
Error  := TRUE;
Busy   := FALSE;
_Error := FALSE;
Status := strStatus;

// Reset 上升緣 → 1 秒閃爍 + retry 觸發 (與 FB_ShippingRobotTransfer 對齊)
trigErrorReset(CLK := Reset);
IF trigErrorReset.Q THEN
	bErrorBlinking := TRUE;
END_IF
tonErrorResetDelay(IN := bErrorBlinking, PT := T#1S);
IF tonErrorResetDelay.Q THEN
	bErrorBlinking := FALSE;
END_IF
IF bErrorBlinking THEN
	Error := FALSE;
END_IF

IF NOT Execute THEN
	Error  := FALSE;
	bErrorBlinking := FALSE;
	tonErrorResetDelay.IN := FALSE;
	eState := STATE_RESETTING;
ELSIF trigErrorReset.Q AND Execute AND NOT Robot._DI1.Error THEN
	// Retry 對稱:Reset 上升緣 (edge) 才觸發,避免 Reset 持續 TRUE 多 cycle 重複切換造成 race
	uiExecutingStep   := uiResumeStep;
	PreviousStrStatus := strStatus;
	PreviousErrorCode := _UniqueErrorCode;
	Status            := 'FB_ShippingPlateScan: no error';
	Error             := FALSE;
	bErrorBlinking    := FALSE;
	tonErrorResetDelay.IN := FALSE;
	_bAbsMoveStarted  := FALSE;	// retry 進 EXECUTING 前清掉,讓 step 3100 ELSIF stale-Done 防護生效
	eState            := STATE_EXECUTING;
END_IF
END_METHOD

METHOD M_STATE_EXECUTING
VAR_INPUT
END_VAR
VAR_INST
	bScanCompleted		: BOOL;		// A2 升 → 已讀 A1 latch,防 A2 transient 重複讀
	bAllowContinue		: BOOL;		// 掃到盒子才 TRUE,送到 _DO3.bContinue 讓手臂繼續夾
END_VAR
Busy := TRUE;

// 暫停
IF Pause THEN
	_HoldingCompleted := FALSE;
	_HeldCompleted    := FALSE;
	_UnholdCompleted  := FALSE;
	uiHoldingStep := 0;
	uiHeldStep    := 0;
	uiUnholdStep  := 0;
	eState := STATE_Holding;
	RETURN;
END_IF

CASE uiExecutingStep OF

	0:	// 命令驗證 + Side→Area + PlateIndex→Address_A
		IF M_ResolveAddress() THEN
			bScanCompleted := FALSE;
			bAllowContinue := FALSE;
			IF __ISVALIDREF(SameSizeCVRequest) THEN
				SameSizeCVRequest.bScan_NeedBackward := FALSE;
			END_IF
			uiExecutingStep := 100;
		ELSE
			Status           := strStatus;
			_UniqueErrorCode := 'E_INVALID_CMD';
			uiResumeStep     := 0;
			_Error := TRUE;
		END_IF

	100:	// Press1 + Press3 一次性伸出 (擋盒避免回流壓到前盒) — 平行處理,兩個都到位才走
			// 用 FB_MachineControl.bSameSizeCV_Press*_AlreadyExtended REFERENCE 做 latch:FALSE → 伸出 + 置 TRUE;TRUE → 跳過
		IF __ISVALIDREF(Cylinder)
		   AND __ISVALIDREF(SameSizeCV_Press1_AlreadyExtended)
		   AND __ISVALIDREF(SameSizeCV_Press3_AlreadyExtended) THEN
			IF SameSizeCV_Press1_AlreadyExtended AND SameSizeCV_Press3_AlreadyExtended THEN
				// 兩個都已 latch,直接跳
				TON_MechTimeOut.IN := FALSE;
				uiExecutingStep := 1000;
			ELSE
				TON_MechTimeOut.IN := TRUE;
				// Press1
				IF NOT SameSizeCV_Press1_AlreadyExtended THEN
					Cylinder.List.fbSameSizeCV_Press1.M_Extend();
					IF Cylinder.List.fbSameSizeCV_Press1.InFrontPosition THEN
						SameSizeCV_Press1_AlreadyExtended := TRUE;
					END_IF
				END_IF
				// Press3
				IF NOT SameSizeCV_Press3_AlreadyExtended THEN
					Cylinder.List.fbSameSizeCV_Press3.M_Extend();
					IF Cylinder.List.fbSameSizeCV_Press3.InFrontPosition THEN
						SameSizeCV_Press3_AlreadyExtended := TRUE;
					END_IF
				END_IF
				// 兩個都到位 → 跳 step 1000
				IF SameSizeCV_Press1_AlreadyExtended AND SameSizeCV_Press3_AlreadyExtended THEN
					TON_MechTimeOut.IN := FALSE;
					uiExecutingStep := 1000;
				END_IF
				IF TON_MechTimeOut.Q THEN
					uiResumeStep := 100;
					strStatus := 'FB_ShippingPlateScan Step 100: Press1/Press3 extend timeout';
					Status := strStatus;
					_UniqueErrorCode := 'E_PRESS_TIMEOUT';
					_Abort := TRUE;
				END_IF
			END_IF
		ELSE
			// ref 無效 (容錯),直接跳到正式流程
			TON_MechTimeOut.IN := FALSE;
			uiExecutingStep := 1000;
		END_IF

	1000:	// 送一次 AbsMove(BoxReady=FALSE) → 手臂走到 safe pos 等 continue 開始掃描
		TON_ScanTimeOut.IN := TRUE;		// 等 A2 掃完旗標 watchdog (給 step 1100 用)

		Robot.M_StartRobotAbsMove(
			GetBox         := TRUE,
			UseClampA      := TRUE,
			UseClampB      := FALSE,
			Area           := Area,
			ClampA_Address := Address_A,
			ClampB_Address := 0,
			BoxReady_1     := FALSE,	// 還沒掃完不下 continue
			BoxReady_2     := FALSE);
		uiExecutingStep := 1100;

		IF Robot._DI1.Error THEN
			uiResumeStep := 1000;
			strStatus := CONCAT('FB_ShippingPlateScan Step 1000: Robot error ', Robot.ErrMsg);
			Status := strStatus;
			_UniqueErrorCode := 'E_ROBOT_ERROR';
			_Abort := TRUE;
		END_IF

	1100:	// 等 A2 (掃描完成旗標) → 讀 A1 latch PlateHasBox (FeedBack 不在這給,做完才給)
		IF Robot.bClampA2_Laser_DetectStatus THEN
			PlateHasBox    := Robot.bClampA1_Laser_DetectStatus;
			bScanCompleted := TRUE;
			TON_ScanTimeOut.IN := FALSE;
			IF NOT PlateHasBox THEN
				// 沒盒 → 跳過取盒/放盒/軌道,直接 step 5000 reset robot 後收尾
				uiExecutingStep := 5000;
			ELSE
				bAllowContinue := TRUE;
				uiExecutingStep := 2000;
			END_IF
		END_IF

		// 早 fail:手臂已 Done 但 A2 從未升起 (Pause 期間手臂跑完命令 / robot prog bug)
		IF Robot._DI1.Done AND NOT bScanCompleted THEN
			uiResumeStep := 1000;
			strStatus := 'FB_ShippingPlateScan Step 1100: Robot done but scan flag (A2) never raised, can retry';
			Status := strStatus;
			_UniqueErrorCode := 'E_SCAN_MISSED';
			_Abort := TRUE;
		END_IF
		IF TON_ScanTimeOut.Q THEN
			uiResumeStep := 1000;	// retry 整個 AbsMove + 掃描流程
			strStatus := 'FB_ShippingPlateScan Step 1100: Scan complete (A2) timeout, can retry';
			Status := strStatus;
			_UniqueErrorCode := 'E_SCAN_TIMEOUT';
			_Abort := TRUE;
		END_IF
		IF Robot._DI1.Error THEN
			uiResumeStep := 1000;
			strStatus := CONCAT('FB_ShippingPlateScan Step 1100: Robot error ', Robot.ErrMsg);
			Status := strStatus;
			_UniqueErrorCode := 'E_ROBOT_ERROR';
			_Abort := TRUE;
		END_IF

	2000:	// 送一次 AbsMove(BoxReady=TRUE) → 手臂收 continue 訊號繼續夾取 → 等 Robot.Done
		TON_RobotActionTimeOut.IN := TRUE;		// 等 Robot.Done watchdog

		Robot.M_StartRobotAbsMove(
			GetBox         := TRUE,
			UseClampA      := TRUE,
			UseClampB      := FALSE,
			Area           := Area,
			ClampA_Address := Address_A,
			ClampB_Address := 0,
			BoxReady_1     := TRUE,		// 下 continue,手臂繼續夾
			BoxReady_2     := FALSE);

		IF Robot._DI1.Done THEN
			TON_RobotActionTimeOut.IN := FALSE;
			uiExecutingStep := 2100;
		END_IF

		IF TON_RobotActionTimeOut.Q THEN
			uiResumeStep := 2000;
			strStatus := 'FB_ShippingPlateScan Step 2000: Robot fetch timeout, can retry';
			Status := strStatus;
			_UniqueErrorCode := 'E_FETCH_TIMEOUT';
			_Abort := TRUE;
		END_IF
		IF Robot._DI1.Error THEN
			uiResumeStep := 2000;
			strStatus := CONCAT('FB_ShippingPlateScan Step 2000: Robot error ', Robot.ErrMsg);
			Status := strStatus;
			_UniqueErrorCode := 'E_ROBOT_ERROR';
			_Abort := TRUE;
		END_IF

	2100:	// Reset FROM AbsMove → 等 Robot.Done 降 (手臂從鐵盤離開準備放盒)
		Robot.M_ResetRobotAbsMove(TRUE, FALSE);
		TON_CheckRobotDoneTimeOut.IN := TRUE;
		IF NOT Robot._DI1.Done THEN
			TON_CheckRobotDoneTimeOut.IN := FALSE;
			uiExecutingStep := 3000;
		END_IF
		IF TON_CheckRobotDoneTimeOut.Q THEN
			uiResumeStep := 2100;
			strStatus := 'FB_ShippingPlateScan Step 2100: Wait Robot done (after fetch) timeout';
			Status := strStatus;
			_UniqueErrorCode := 'E_ROBOT_DONE_TIMEOUT';
			_Error := TRUE;
		END_IF

	// ===========================================================
	// Phase 2 (TO):放盒到同尺寸軌道 TransmitCV_End Pos 1 SameSize
	// 對齊 FB_ShippingRobotTransfer step 10300/15000/15100/20000
	// ===========================================================
	3000:	// TO 前置:請求 backward (arbiter 驅動) + 等放盒位 sensor 清空
		IF __ISVALIDREF(SameSizeCVRequest) THEN
			SameSizeCVRequest.bScan_NeedBackward := TRUE;
		END_IF
		TON_MechTimeOut.IN := TRUE;
		IF __ISVALIDREF(Motor) AND Motor.List.TransmitSameSideCV.InBackWard
		   AND NOT Input.bSameSizeCV_BoxNearShippingSensor THEN
			TON_MechTimeOut.IN := FALSE;
			uiExecutingStep := 3100;
		END_IF
		IF TON_MechTimeOut.Q THEN
			uiResumeStep := 3000;
			strStatus := 'FB_ShippingPlateScan Step 3000: SameSizeCV backward / sensor clear timeout';
			Status := strStatus;
			_UniqueErrorCode := 'E_CV_BACKWARD_TIMEOUT';
			_Abort := TRUE;
		END_IF

	3100:	// AbsMove 到 TransmitCV_End Pos 1 放盒
			// Put 場景:step 3000 已驗證軌道反轉 + sensor 清,BoxReady 直接 TRUE (對齊 FB_ShippingRobotTransfer 15000 Put 分支)
			// _bAbsMoveStarted 防 ghost completion:step 2100 ResetAbsMove 後 Done 可能殘留 TRUE
		TON_RobotActionTimeOut.IN := TRUE;
		IF NOT Robot._DI1.Done THEN
			Robot.M_StartRobotAbsMove(
				GetBox         := FALSE,
				UseClampA      := TRUE,
				UseClampB      := FALSE,
				Area           := E_RobotArea.TransmitCV_End,
				ClampA_Address := 1,
				ClampB_Address := 0,
				BoxReady_1     := TRUE,
				BoxReady_2     := FALSE);
			_bAbsMoveStarted := TRUE;
		ELSIF NOT _bAbsMoveStarted THEN
			// Done=TRUE 但從未送過 Start → stale (step 2100 殘留),清掉 robot 命令等 Done 降
			Robot.M_ResetRobotAbsMove(TRUE, FALSE);
		ELSE
			// 真的完成 (Done 從 FALSE → TRUE)
			TON_RobotActionTimeOut.IN := FALSE;
			_bAbsMoveStarted          := FALSE;
			uiExecutingStep := 3200;
		END_IF

		IF TON_RobotActionTimeOut.Q THEN
			uiResumeStep := 3100;
			strStatus := 'FB_ShippingPlateScan Step 3100: Robot put to SameSizeCV timeout';
			Status := strStatus;
			_UniqueErrorCode := 'E_PUT_TIMEOUT';
			_Abort := TRUE;
		END_IF
		IF Robot._DI1.Error THEN
			uiResumeStep := 3100;
			strStatus := CONCAT('FB_ShippingPlateScan Step 3100: Robot error ', Robot.ErrMsg);
			Status := strStatus;
			_UniqueErrorCode := 'E_ROBOT_ERROR';
			_Abort := TRUE;
		END_IF

	3200:	// Reset TO AbsMove → 等 Robot.Done 降
		Robot.M_ResetRobotAbsMove(TRUE, FALSE);
		TON_CheckRobotDoneTimeOut.IN := TRUE;
		IF NOT Robot._DI1.Done THEN
			TON_CheckRobotDoneTimeOut.IN := FALSE;
			uiExecutingStep := 3300;
		END_IF
		IF TON_CheckRobotDoneTimeOut.Q THEN
			uiResumeStep := 3200;
			strStatus := 'FB_ShippingPlateScan Step 3200: Wait Robot done (after put) timeout';
			Status := strStatus;
			_UniqueErrorCode := 'E_ROBOT_DONE_TIMEOUT';
			_Error := TRUE;
		END_IF

	3300:	// TO 後置:確保 backward 持續請求 (推走剛放的盒子,arbiter 驅動)
		IF __ISVALIDREF(SameSizeCVRequest) THEN
			SameSizeCVRequest.bScan_NeedBackward := TRUE;
		END_IF
		uiExecutingStep := 3400;

	3400:	// 等馬達 backward 起步 → 進 FeedBack (軌道不停,持續推到 STATE_DONE 才停)
		TON_MechTimeOut.IN := TRUE;
		IF __ISVALIDREF(Motor) AND Motor.List.TransmitSameSideCV.InBackWard THEN
			TON_MechTimeOut.IN := FALSE;
			uiExecutingStep := 4000;
		END_IF
		IF TON_MechTimeOut.Q THEN
			uiResumeStep := 3400;
			strStatus := 'FB_ShippingPlateScan Step 3400: SameSizeCV backward timeout';
			Status := strStatus;
			_UniqueErrorCode := 'E_CV_BACKWARD_TIMEOUT';
			_Abort := TRUE;
		END_IF

	// ===========================================================
	// 沒盒 path:跳過取盒/放盒/軌道,直接 reset robot 進收尾
	// ===========================================================
	5000:	// Reset robot 命令 → 等 Done 降 (沒盒專用)
		Robot.M_ResetRobotAbsMove(TRUE, FALSE);
		TON_CheckRobotDoneTimeOut.IN := TRUE;
		IF NOT Robot._DI1.Done AND Robot.M_CheckResetAllCommand() THEN
			TON_CheckRobotDoneTimeOut.IN := FALSE;
			uiExecutingStep := 5100;
		END_IF
		IF TON_CheckRobotDoneTimeOut.Q THEN
			uiResumeStep := 5000;
			strStatus := 'FB_ShippingPlateScan Step 5000: Wait Robot done (no box) timeout';
			Status := strStatus;
			_UniqueErrorCode := 'E_ROBOT_DONE_TIMEOUT';
			_Error := TRUE;
		END_IF
		
	5100:
		TON_CheckRobotDoneTimeOut.IN := TRUE;
		TON_RobotCommandDelay.IN     := TRUE;
		IF  NOT PlateHasBox THEN				//檢查是否是第四盒且沒有盒子
			IF TON_RobotCommandDelay.Q THEN
				IF Robot.M_ReleaseRobotInternalCycle() THEN		// 給手臂清除流程命令。
					uiExecutingStep := 5200;
				END_IF
			END_IF
		ELSE
			uiExecutingStep := 4000;
		END_IF
		IF TON_CheckRobotDoneTimeOut.Q THEN
			uiResumeStep := 5100;
			strStatus := 'FB_ShippingPlateScan Step 5100: Send Robot Clear Internal Cylce Timeout';
			Status := strStatus;
			_UniqueErrorCode := 'E_ROBOT_DONE_TIMEOUT';
			_Error := TRUE;
		END_IF
		
	5200:
		IF Robot._DI1.Done THEN
			IF Robot.M_ResetInternalCycleCommand() THEN
				uiExecutingStep := 5300;
			END_IF
		END_IF
	
	5300:
		Robot.M_ResetInternalCycleCommand() ;
		IF NOT Robot._DI1.Done THEN
			uiExecutingStep := 4000;
		END_IF

	// ===========================================================
	// 收尾:做完才給 FeedBack → 等 ReadComplete → 清 FeedBack
	// ===========================================================
	4000:	// 整個動作完成 → FeedBack:=TRUE 通知上位讀 PlateHasBox
		FeedBack := TRUE;
		IF ReadComplete THEN
			FeedBack := FALSE;
			uiExecutingStep := 90000;
		END_IF

	90000:
		Status    := 'FB_ShippingPlateScan: Process completed';
		_Executed := TRUE;
END_CASE

// 狀態機切換
IF NOT Execute THEN
	eState := STATE_RESETTING;
ELSIF _Error THEN
	eState := STATE_ERROR;
ELSIF _Abort THEN
	eState := STATE_ABORTING;
ELSIF _Executed THEN
	eState := STATE_DONE;
END_IF
END_METHOD

METHOD M_STATE_HELD
VAR_INPUT
END_VAR
Busy   := FALSE;
Paused := TRUE;

CASE uiHeldStep OF
	0:
		uiHeldStep := 9999;
	9999:
		_HeldCompleted := TRUE;
END_CASE

IF _HeldCompleted AND NOT Pause THEN
	eState := STATE_UnHold;
END_IF
END_METHOD

METHOD M_STATE_HOLDING
VAR_INPUT
END_VAR
CASE uiHoldingStep OF
	0:
		TON_RobotActionTimeOut.IN    := FALSE;
		TON_CheckRobotDoneTimeOut.IN := FALSE;
		TON_ScanTimeOut.IN           := FALSE;
		uiHoldingStep := 9999;
	9999:
		_HoldingCompleted := TRUE;
END_CASE

IF _HoldingCompleted THEN
	eState := STATE_Held;
END_IF
END_METHOD

METHOD M_STATE_RESETTING
VAR_INPUT
END_VAR
CASE uiResettingStep OF
	0:
		TON_RobotActionTimeOut.IN    := FALSE;
		TON_CheckRobotDoneTimeOut.IN := FALSE;
		TON_ScanTimeOut.IN           := FALSE;
		TON_MechTimeOut.IN           := FALSE;
		tonBoxArriveDelay.IN         := FALSE;
		TON_RobotCommandDelay.IN	 := FALSE;
		// 撤銷軌道請求 (arbiter 看到沒人 request 會自動停)
		IF __ISVALIDREF(SameSizeCVRequest) THEN
			SameSizeCVRequest.bScan_NeedBackward := FALSE;
		END_IF
		_bAbsMoveStarted := FALSE;
		PlateHasBox := FALSE;
		FeedBack    := FALSE;
		uiResettingStep := 100;

	100:
		Robot.M_ResetAllCommand();
		IF Robot.M_CheckResetAllCommand() AND Robot.M_ResetInternalCycleCommand()THEN
			uiResettingStep := 9999;
		END_IF

	9999:
		_ResetCompleted := TRUE;
END_CASE

IF _ResetCompleted THEN
	eState := STATE_DORMANT;
END_IF
END_METHOD

METHOD M_STATE_UNHOLD
VAR_INPUT
END_VAR
CASE uiUnholdStep OF
	0:
		uiUnholdStep := 9999;
	9999:
		_UnholdCompleted := TRUE;
END_CASE

IF _UnholdCompleted THEN
	Paused := FALSE;
	eState := STATE_EXECUTING;
END_IF
END_METHOD

END_FUNCTION_BLOCK

// ---- Library/20_MachineUnits/23_ShippingArea/Service/FB_ShippingTransCV_LeftSide.TcPOU
FUNCTION_BLOCK FB_ShippingTransCV_LeftSide EXTENDS FB_ActionBasic
VAR_INPUT
    xExecute    : BOOL;
    xAbort      : BOOL;
	xReset		: BOOL;
	TimeOut  	: LREAL := 60; // Unit : s
    Cylinder 	: REFERENCE TO UNI_CylinderList;
	Motor		: REFERENCE TO UNI_MotorList;
	Input		: REFERENCE TO ST_InputTable;
	OutPut		: REFERENCE TO ST_OutputTable;
	ShippingTransCVRequest_LeftSide : BOOL;
	RobotStatus	: ST_StatusBasic;		// robot Service 
END_VAR
VAR_OUTPUT
	xAborted : BOOL;
    iErrorID : INT;
    ErrorMsg : STRING;
END_VAR
VAR
	// model setting 
	StateBehaviour   : CBML.ETrigATo;
    CurrentPosition : ST_PositionTable;
	fbExecuteEdgeDetect :FB_EdgeDetect;
	Reset_Rtrig 	:R_TRIG;
	uiCyclicStep    : UINT := 0;
	
	//Timer
	TON_DelayArrivedDetect	: TON;
	TON_TransCVAllowDelay	: TON;
END_VAR

THIS^.IBehaviourModel := StateBehaviour;

StateBehaviour(xExecute := xExecute,
              xAbort := xAbort OR fbExecuteEdgeDetect.xFallingEdge,
              udiTimeOut := LREAL_TO_UDINT( TimeOut*1000000),
              xDone => xDone,
              xBusy => xBusy,
              xError => xError,
              xAborted => xAborted);
			  
//Make sure that C# turns off execute to shut down the service
fbExecuteEdgeDetect(xInput :=xExecute);
  
//Error Msg
iErrorID := StateBehaviour._model.iErrorID;
ErrorMsg := M_GetErrorMsg(xErrorID := iErrorID);

//Reset
Reset_Rtrig(CLK:= xReset);
IF Reset_Rtrig.Q THEN
	StateBehaviour.ResetModel(xCommit:=xReset);
END_IF

//Action
A00_BaseUnit();

ACTION A00_BaseUnit:
TON_DelayArrivedDetect(PT:=T#1S);
TON_TransCVAllowDelay(PT :=T#1S);
END_ACTION

METHOD CleanupAction
VAR_INPUT
    xAbortProposed : BOOL;
    iErrorIDProposed: INT;
END_VAR
VAR_OUTPUT
    xComplete : BOOL := TRUE;
    xAbort: BOOL := xAbortProposed;
 	iErrorID : INT := iErrorIDProposed;
END_VAR
END_METHOD

METHOD CyclicAction
VAR_INPUT
    itfTimingController : CBML.ITimingController;
END_VAR
VAR_OUTPUT
    xComplete : BOOL := TRUE;
    iErrorID : INT := 0;
END_VAR
xComplete := FALSE;


CASE uiCyclicStep OF 
	0:	// robot status , send allow signal
		IF ShippingTransCVRequest_LeftSide AND NOT RobotStatus.Busy THEN
			TON_TransCVAllowDelay.IN := TRUE;
			OutPut.bShippingTransCV_Leftside_Allow := TRUE;
		END_IF
		IF TON_TransCVAllowDelay.Q THEN
			OutPut.bShippingTransCV_Leftside_Allow := FALSE;
			uiCyclicStep := 100;
		END_IF

	100:	//check HansLaser cancel signal
		TON_TransCVAllowDelay.IN := FALSE;
		IF NOT Input.bShippingTransCV_Leftside_Arrived THEN 
			xComplete := TRUE;
		END_IF
END_CASE

IF Input.bHansLaserMachineError THEN
	iErrorID := 10;
END_IF
END_METHOD

METHOD ExitAction
VAR_INPUT
    xAfterCleanup : BOOL;
    xInCopyCode : BOOL;
END_VAR
END_METHOD

METHOD M_GetErrorMsg : T_MaxString
VAR_INPUT
	xErrorID: INT;
END_VAR

VAR
	
END_VAR
CASE xErrorID OF
	0:
		M_GetErrorMsg := 'No Error';
	1:
		M_GetErrorMsg := 'FB_ShippingTransCV_LeftSide ErrorID 1: Action time out';
///
	10:
		M_GetErrorMsg := 'FB_ShippingTransCV_LeftSide ErrorID 10: HansLaser Machine Error';
	11:
		M_GetErrorMsg := 'FB_ShippingTransCV_LeftSide ErrorID 11: Wrong Command , TransCV not IntargetPosition';
END_CASE
END_METHOD

METHOD ResetAction
VAR_OUTPUT
    xComplete : BOOL := TRUE;
END_VAR
xComplete := FALSE;

ShippingTransCVRequest_LeftSide 		:= FALSE;
OutPut.bShippingTransCV_Leftside_Allow := FALSE;

TON_DelayArrivedDetect.IN := FALSE;
TON_TransCVAllowDelay.IN := FALSE;

uiCyclicStep := 0;

xComplete := TRUE;
END_METHOD

METHOD StartAction
VAR_OUTPUT
    xComplete : BOOL := TRUE;
	iErrorID : INT := 0;
END_VAR
xComplete := FALSE;

ShippingTransCVRequest_LeftSide 		:= FALSE;
OutPut.bShippingTransCV_Leftside_Allow := FALSE;

uiCyclicStep := 0;

TON_DelayArrivedDetect.IN := FALSE;
TON_TransCVAllowDelay.IN := FALSE;


xComplete := TRUE;

IF Input.bHansLaserMachineError THEN
	iErrorID := 10;
END_IF

IF NOT Input.bShippingTransCV_Leftside_Arrived THEN
	iErrorID := 11;
END_IF
END_METHOD

END_FUNCTION_BLOCK

// ---- Library/20_MachineUnits/23_ShippingArea/Service/FB_ShippingTransCV_RightSide.TcPOU
FUNCTION_BLOCK FB_ShippingTransCV_RightSide EXTENDS FB_ActionBasic
VAR_INPUT
    xExecute    : BOOL;
    xAbort      : BOOL;
	xReset		: BOOL;
	TimeOut  	: LREAL := 60; // Unit : s
    Cylinder 	: REFERENCE TO UNI_CylinderList;
	Motor		: REFERENCE TO UNI_MotorList;
	Input		: REFERENCE TO ST_InputTable;
	OutPut		: REFERENCE TO ST_OutputTable;
	ShippingTransCVRequest_RightSide : BOOL;
	RobotStatus	: ST_StatusBasic;		// robot Service 
END_VAR
VAR_OUTPUT
	xAborted : BOOL;
    iErrorID : INT;
    ErrorMsg : STRING;
END_VAR
VAR
	// model setting 
	StateBehaviour   : CBML.ETrigATo;
    CurrentPosition : ST_PositionTable;
	fbExecuteEdgeDetect :FB_EdgeDetect;
	Reset_Rtrig 	:R_TRIG;
	uiCyclicStep    : UINT := 0;
	
	//Timer
	TON_DelayArrivedDetect	: TON;
	TON_TransCVAllowDelay	: TON;
END_VAR

THIS^.IBehaviourModel := StateBehaviour;

StateBehaviour(xExecute := xExecute,
              xAbort := xAbort OR fbExecuteEdgeDetect.xFallingEdge,
              udiTimeOut := LREAL_TO_UDINT( TimeOut*1000000),
              xDone => xDone,
              xBusy => xBusy,
              xError => xError,
              xAborted => xAborted);
			  
//Make sure that C# turns off execute to shut down the service
fbExecuteEdgeDetect(xInput :=xExecute);
  
//Error Msg
iErrorID := StateBehaviour._model.iErrorID;
ErrorMsg := M_GetErrorMsg(xErrorID := iErrorID);

//Reset
Reset_Rtrig(CLK:= xReset);
IF Reset_Rtrig.Q THEN
	StateBehaviour.ResetModel(xCommit:=xReset);
END_IF

//Action
A00_BaseUnit();

ACTION A00_BaseUnit:
TON_DelayArrivedDetect(PT:=T#1S);
TON_TransCVAllowDelay(PT :=T#1S);
END_ACTION

METHOD CleanupAction
VAR_INPUT
    xAbortProposed : BOOL;
    iErrorIDProposed: INT;
END_VAR
VAR_OUTPUT
    xComplete : BOOL := TRUE;
    xAbort: BOOL := xAbortProposed;
 	iErrorID : INT := iErrorIDProposed;
END_VAR
END_METHOD

METHOD CyclicAction
VAR_INPUT
    itfTimingController : CBML.ITimingController;
END_VAR
VAR_OUTPUT
    xComplete : BOOL := TRUE;
    iErrorID : INT := 0;
END_VAR
xComplete := FALSE;


CASE uiCyclicStep OF 
	0:	// robot status , send allow signal
		IF ShippingTransCVRequest_RightSide AND NOT RobotStatus.Busy THEN
			TON_TransCVAllowDelay.IN := TRUE;
			OutPut.bShippingTransCV_Rightside_Allow := TRUE;
		END_IF
		IF TON_TransCVAllowDelay.Q THEN
			OutPut.bShippingTransCV_Rightside_Allow := FALSE;
			uiCyclicStep := 100;
		END_IF

	100:	//check HansLaser cancel signal
		TON_TransCVAllowDelay.IN := FALSE;
		IF NOT Input.bShippingTransCV_Rightside_Arrived THEN 
			xComplete := TRUE;
		END_IF
END_CASE

IF Input.bHansLaserMachineError THEN
	iErrorID := 10;
END_IF
END_METHOD

METHOD ExitAction
VAR_INPUT
    xAfterCleanup : BOOL;
    xInCopyCode : BOOL;
END_VAR
END_METHOD

METHOD M_GetErrorMsg : T_MaxString
VAR_INPUT
	xErrorID: INT;
END_VAR

VAR
	
END_VAR
CASE xErrorID OF
	0:
		M_GetErrorMsg := 'No Error';
	1:
		M_GetErrorMsg := 'FB_ShippingTransCV_RightSide ErrorID 1: Action time out';
///
	10:
		M_GetErrorMsg := 'FB_ShippingTransCV_RightSide ErrorID 10: HansLaser Machine Error';
	11:
		M_GetErrorMsg := 'FB_ShippingTransCV_RightSide ErrorID 11: Wrong Command , TransCV not IntargetPosition';
END_CASE
END_METHOD

METHOD ResetAction
VAR_OUTPUT
    xComplete : BOOL := TRUE;
END_VAR
xComplete := FALSE;

ShippingTransCVRequest_RightSide 		:= FALSE;
OutPut.bShippingTransCV_Rightside_Allow := FALSE;

TON_DelayArrivedDetect.IN := FALSE;
TON_TransCVAllowDelay.IN := FALSE;

uiCyclicStep := 0;

xComplete := TRUE;
END_METHOD

METHOD StartAction
VAR_OUTPUT
    xComplete : BOOL := TRUE;
	iErrorID : INT := 0;
END_VAR
xComplete := FALSE;

ShippingTransCVRequest_RightSide 		:= FALSE;
OutPut.bShippingTransCV_Rightside_Allow := FALSE;

uiCyclicStep := 0;

TON_DelayArrivedDetect.IN := FALSE;
TON_TransCVAllowDelay.IN := FALSE;




IF Input.bHansLaserMachineError THEN
	iErrorID := 10;
END_IF

IF NOT Input.bShippingTransCV_Rightside_Arrived THEN
	iErrorID := 11;
END_IF

xComplete := TRUE;
END_METHOD

END_FUNCTION_BLOCK

// ---- Library/99_Utilities/FB_TableMove.TcPOU
FUNCTION_BLOCK FB_TableMove EXTENDS FB_ActionBasic
VAR_INPUT
    xExecute    : BOOL;
    xAbort      : BOOL;
    xReset      : BOOL;
    Index       : INT; // PositionTable array index
    CurrentData : REFERENCE TO ST_SetupPara; // Componets setup parameter
    TimeOut     : LREAL := 30; // Unit : s
END_VAR
VAR_OUTPUT
    xAborted : BOOL;
    iErrorID : INT;
    ErrorMsg : T_MaxString;
END_VAR
VAR
    // State Machine
    StateBehaviour  : CBML.ETrigATo;
    CurrentPosition : ST_PositionTable;
	
	Cylinder : UNI_CylinderList;
	Reset_Rtrig : R_TRIG;
	fbExecuteEdgeDetect :FB_EdgeDetect;
END_VAR

THIS^.IBehaviourModel := StateBehaviour;
StateBehaviour(xExecute := xExecute,
               xAbort := xAbort OR fbExecuteEdgeDetect.xFallingEdge,
               udiTimeOut := LREAL_TO_UDINT( TimeOut*1000000),
               xDone => xDone,
               xBusy => xBusy,
               xError => xError,
               xAborted => xAborted);

//Error Msg
iErrorID := StateBehaviour._model.iErrorID;
ErrorMsg := M_GetErrorMsg(xErrorID := iErrorID);

//Make sure that C# turns off execute to shut down the service
fbExecuteEdgeDetect(xInput :=xExecute);

//Reset
Reset_Rtrig(CLK:= xReset);
IF Reset_Rtrig.Q THEN
	StateBehaviour.ResetModel(xCommit:=xReset);
END_IF

METHOD CleanupAction
VAR_INPUT
    xAbortProposed : BOOL;
    iErrorIDProposed: INT;
END_VAR
VAR_OUTPUT
    xComplete : BOOL := TRUE;
    xAbort: BOOL := xAbortProposed;
 	iErrorID : INT := iErrorIDProposed;
END_VAR
END_METHOD

METHOD CyclicAction
VAR_INPUT
    itfTimingController : CBML.ITimingController;
END_VAR
VAR_OUTPUT
    xComplete : BOOL := TRUE;
    iErrorID : INT := 0;
END_VAR
VAR_INST
	AllowAllocateRobotMove : BOOL;
	AllowOutRobotMove : BOOL;
	AllowRoundBeltMove : BOOL;
	AllowTurnTable :BOOL;
END_VAR
///safe check

xComplete := FALSE;
IF CurrentPosition.Robot = 1  THEN
	arAxisCtrl_gb[AxisNo.OutRobot_X].PosMode.Acc := CurrentData.Axes.OutRobot_X.HalfAuto.Acceleration;
	arAxisCtrl_gb[AxisNo.OutRobot_X].PosMode.Dec := CurrentData.Axes.OutRobot_X.HalfAuto.Deceleration;
	arAxisCtrl_gb[AxisNo.OutRobot_X].PosMode.Jerk := CurrentData.Axes.OutRobot_X.HalfAuto.Jerk;
	arAxisCtrl_gb[AxisNo.OutRobot_X].PosMode.Velocity := CurrentData.Axes.OutRobot_X.HalfAuto.Velocity;
	arAxisCtrl_gb[AxisNo.OutRobot_X].PosMode.Position := CurrentPosition.X_Pos;

	arAxisCtrl_gb[AxisNo.OutRobot_Y].PosMode.Acc := CurrentData.Axes.OutRobot_X.HalfAuto.Acceleration;
	arAxisCtrl_gb[AxisNo.OutRobot_Y].PosMode.Dec := CurrentData.Axes.OutRobot_X.HalfAuto.Deceleration;
	arAxisCtrl_gb[AxisNo.OutRobot_Y].PosMode.Jerk := CurrentData.Axes.OutRobot_X.HalfAuto.Jerk;
	arAxisCtrl_gb[AxisNo.OutRobot_Y].PosMode.Velocity := CurrentData.Axes.OutRobot_X.HalfAuto.Velocity;
	arAxisCtrl_gb[AxisNo.OutRobot_Y].PosMode.Position := CurrentPosition.Y_Pos;
	IF arAxisStatus_gb[AxisNo.OutRobot_X].Admin._OpModeAck = ModePosAbs AND arAxisStatus_gb[AxisNo.OutRobot_X].Admin.CmdDone AND 
		arAxisStatus_gb[AxisNo.OutRobot_Y].Admin._OpModeAck = ModePosAbs AND arAxisStatus_gb[AxisNo.OutRobot_Y].Admin.CmdDone THEN
		xComplete := TRUE;
	END_IF

ELSIF CurrentPosition.Robot = 0  THEN
	arAxisCtrl_gb[AxisNo.Allocate_X].PosMode.Acc := CurrentData.Axes.Allocate_X.HalfAuto.Acceleration;
	arAxisCtrl_gb[AxisNo.Allocate_X].PosMode.Dec := CurrentData.Axes.Allocate_X.HalfAuto.Deceleration;
	arAxisCtrl_gb[AxisNo.Allocate_X].PosMode.Jerk := CurrentData.Axes.Allocate_X.HalfAuto.Jerk;
	arAxisCtrl_gb[AxisNo.Allocate_X].PosMode.Velocity := CurrentData.Axes.Allocate_X.HalfAuto.Velocity;
	arAxisCtrl_gb[AxisNo.Allocate_X].PosMode.Position := CurrentPosition.X_Pos;

	arAxisCtrl_gb[AxisNo.Allocate_Y].PosMode.Acc := CurrentData.Axes.Allocate_Y.HalfAuto.Acceleration;
	arAxisCtrl_gb[AxisNo.Allocate_Y].PosMode.Dec := CurrentData.Axes.Allocate_Y.HalfAuto.Deceleration;
	arAxisCtrl_gb[AxisNo.Allocate_Y].PosMode.Jerk := CurrentData.Axes.Allocate_Y.HalfAuto.Jerk;
	arAxisCtrl_gb[AxisNo.Allocate_Y].PosMode.Velocity := CurrentData.Axes.Allocate_Y.HalfAuto.Velocity;
	arAxisCtrl_gb[AxisNo.Allocate_Y].PosMode.Position := CurrentPosition.Y_Pos;
	IF arAxisStatus_gb[AxisNo.Allocate_X].Admin._OpModeAck = ModePosAbs AND arAxisStatus_gb[AxisNo.Allocate_X].Admin.CmdDone AND 
		arAxisStatus_gb[AxisNo.Allocate_Y].Admin._OpModeAck = ModePosAbs AND arAxisStatus_gb[AxisNo.Allocate_Y].Admin.CmdDone THEN
		xComplete := TRUE;
	END_IF

ELSIF CurrentPosition.Robot = 2  THEN
	arAxisCtrl_gb[AxisNo.RoundBelt].PosMode.Acc := CurrentData.Axes.RoundBelt.HalfAuto.Acceleration;
	arAxisCtrl_gb[AxisNo.RoundBelt].PosMode.Dec := CurrentData.Axes.RoundBelt.HalfAuto.Deceleration;
	arAxisCtrl_gb[AxisNo.RoundBelt].PosMode.Jerk := CurrentData.Axes.RoundBelt.HalfAuto.Jerk;
	arAxisCtrl_gb[AxisNo.RoundBelt].PosMode.Velocity := CurrentData.Axes.RoundBelt.HalfAuto.Velocity;
	arAxisCtrl_gb[AxisNo.RoundBelt].PosMode.Position := CurrentPosition.X_Pos;
	IF arAxisStatus_gb[AxisNo.RoundBelt].Admin._OpModeAck = ModePosAbs AND arAxisStatus_gb[AxisNo.RoundBelt].Admin.CmdDone  THEN
		xComplete := TRUE;
	END_IF

ELSIF CurrentPosition.Robot = 3 THEN
	arAxisCtrl_gb[AxisNo.TurnTable].PosMode.Acc := CurrentData.Axes.TurnTable.HalfAuto.Acceleration;
	arAxisCtrl_gb[AxisNo.TurnTable].PosMode.Dec := CurrentData.Axes.TurnTable.HalfAuto.Deceleration;
	arAxisCtrl_gb[AxisNo.TurnTable].PosMode.Jerk := CurrentData.Axes.TurnTable.HalfAuto.Jerk;
	arAxisCtrl_gb[AxisNo.TurnTable].PosMode.Velocity := CurrentData.Axes.TurnTable.HalfAuto.Velocity;
	arAxisCtrl_gb[AxisNo.TurnTable].PosMode.Position := CurrentPosition.X_Pos;
	IF arAxisStatus_gb[AxisNo.TurnTable].Admin._OpModeAck = ModePosAbs AND arAxisStatus_gb[AxisNo.TurnTable].Admin.CmdDone  THEN
		xComplete := TRUE;
	END_IF

ELSIF CurrentPosition.Robot = 4 THEN
	arAxisCtrl_gb[AxisNo.RackMotor].PosMode.Acc := CurrentData.Axes.RackMotor.HalfAuto.Acceleration;
	arAxisCtrl_gb[AxisNo.RackMotor].PosMode.Dec := CurrentData.Axes.RackMotor.HalfAuto.Deceleration;
	arAxisCtrl_gb[AxisNo.RackMotor].PosMode.Jerk := CurrentData.Axes.RackMotor.HalfAuto.Jerk;
	arAxisCtrl_gb[AxisNo.RackMotor].PosMode.Velocity := CurrentData.Axes.RackMotor.HalfAuto.Velocity;
	arAxisCtrl_gb[AxisNo.RackMotor].PosMode.Position := CurrentPosition.X_Pos;
	IF arAxisStatus_gb[AxisNo.RackMotor].Admin._OpModeAck = ModePosAbs AND arAxisStatus_gb[AxisNo.RackMotor].Admin.CmdDone  THEN
		xComplete := TRUE;
	END_IF

END_IF

IF arAxisCtrl_gb[AxisNo.OutRobot_X].Admin.Axis.Status.Error THEN
	iErrorID := 5; // Axis OutRobot_X has error
END_IF
IF arAxisCtrl_gb[AxisNo.OutRobot_Y].Admin.Axis.Status.Error THEN
	iErrorID := 6; // Axis OutRobotY has error
END_IF
IF arAxisCtrl_gb[AxisNo.Allocate_X].Admin.Axis.Status.Error THEN
	iErrorID := 7; // Axis Allocate_X has error
END_IF
IF arAxisCtrl_gb[AxisNo.Allocate_Y].Admin.Axis.Status.Error THEN
	iErrorID := 8; // Axis Allocate_Y has error
END_IF
IF arAxisCtrl_gb[AxisNo.RoundBelt].Admin.Axis.Status.Error THEN
	iErrorID := 9; // Axis RoundBelt has error
END_IF
IF arAxisCtrl_gb[AxisNo.TurnTable].Admin.Axis.Status.Error THEN
	iErrorID := 10; // Axis TurnTable has error
END_IF
END_METHOD

METHOD ExitAction
VAR_INPUT
    xAfterCleanup : BOOL;
    xInCopyCode : BOOL;
END_VAR
END_METHOD

METHOD M_GetErrorMsg : T_MaxString
VAR_INPUT
	xErrorID: INT;
END_VAR

VAR
	
END_VAR
CASE xErrorID OF
    0:
        M_GetErrorMsg := 'No Error';
    1:
        M_GetErrorMsg := 'FB_TableMove ErrorID 1: Action time out';
    2:
        M_GetErrorMsg := 'FB_TableMove ErrorID 2: Position Data invalid';
    3:
        M_GetErrorMsg := 'FB_TableMove ErrorID 3: Index invalid';
    4:
		M_GetErrorMsg := 'FB_TableMove ErrorID 4: Axis is not ready';
    5:
        M_GetErrorMsg := 'FB_TableMove ErrorID 5: Axis OutRobot X has Error';
    6:
        M_GetErrorMsg := 'FB_TableMove ErrorID 6: Axis OutRobot Y has Error';
	7:
		M_GetErrorMsg := 'FB_TableMove ErrorID 7: Axis Allocate_X has error';
	8:
		M_GetErrorMsg := 'FB_TableMove ErrorID 8: Axis Allocate_Y has error';
	9:
		M_GetErrorMsg := 'FB_TableMove ErrorID 9: Axis RoundBelt has error';
	10:
		M_GetErrorMsg := 'FB_TableMove ErrorID 10: Axis TurnTable has error';
END_CASE
END_METHOD

METHOD ResetAction
VAR_OUTPUT
    xComplete : BOOL := TRUE;
END_VAR
END_METHOD

METHOD StartAction
VAR_OUTPUT
    xComplete : BOOL := TRUE;
	iErrorID : INT := 0;
END_VAR
IF Index >= 1 AND Index <= 200 THEN
CurrentPosition := CurrentData.PositionTable[Index];
ELSE
	iErrorID := 3; // Index invalid
	RETURN;
END_IF
//0 : Allocate , 1: OutRobot, 2: RoundBelt , 3: TurnTable, 4: RackMotor
IF CurrentPosition.Robot = 1  THEN		
	IF arAxisCtrl_gb[AxisNo.OutRobot_X].Admin.Axis.Status.NotMoving AND  
		NOT arAxisCtrl_gb[AxisNo.OutRobot_X].Admin.Axis.Status.Error AND 
		arAxisCtrl_gb[AxisNo.OutRobot_Y].Admin.Axis.Status.NotMoving AND
		NOT arAxisCtrl_gb[AxisNo.OutRobot_Y].Admin.Axis.Status.Error
		THEN
		xComplete := TRUE;
	ELSE
		iErrorID := 4; // Axis not ready
	END_IF
ELSIF CurrentPosition.Robot = 0  THEN
	IF arAxisCtrl_gb[AxisNo.Allocate_X].Admin.Axis.Status.NotMoving AND  
		NOT arAxisCtrl_gb[AxisNo.Allocate_X].Admin.Axis.Status.Error AND 
		arAxisCtrl_gb[AxisNo.Allocate_Y].Admin.Axis.Status.NotMoving AND
		NOT arAxisCtrl_gb[AxisNo.Allocate_Y].Admin.Axis.Status.Error
		THEN
		xComplete := TRUE;
	ELSE
		iErrorID := 4; // Axis not ready
	END_IF
ELSIF CurrentPosition.Robot = 2  THEN
	IF arAxisCtrl_gb[AxisNo.RoundBelt].Admin.Axis.Status.NotMoving AND  
		NOT arAxisCtrl_gb[AxisNo.RoundBelt].Admin.Axis.Status.Error THEN
		xComplete := TRUE;
	ELSE
		iErrorID := 4; // Axis not ready
	END_IF
ELSIF CurrentPosition.Robot = 3  THEN
	IF arAxisCtrl_gb[AxisNo.TurnTable].Admin.Axis.Status.NotMoving AND  
		NOT arAxisCtrl_gb[AxisNo.TurnTable].Admin.Axis.Status.Error THEN 
		xComplete := TRUE;
	ELSE
		iErrorID := 4; // Axis not ready
	END_IF
ELSIF CurrentPosition.Robot = 4  THEN
	IF arAxisCtrl_gb[AxisNo.RackMotor].Admin.Axis.Status.NotMoving AND  
		NOT arAxisCtrl_gb[AxisNo.RackMotor].Admin.Axis.Status.Error THEN 
		xComplete := TRUE;
	ELSE
		iErrorID := 4; // Axis not ready
	END_IF
ELSE
	iErrorID := 2; // Position Data invalid
END_IF
END_METHOD

END_FUNCTION_BLOCK

// ---- Library/10_Machine/12_MachineControl/Service/FB_MachineHoming.TcPOU
FUNCTION_BLOCK FB_MachineHoming EXTENDS FB_ActionBasic
VAR_INPUT
	xExecute : BOOL;
	xAbort : BOOL;
    AllocateHome : REFERENCE TO  FB_AllocateAreaHome;
    StorageHome  :REFERENCE TO FB_StorageHoming;
    ShippingHome :REFERENCE TO FB_ShippingHoming;
	AllocateHomed : REFERENCE TO BOOL;
	StorageHomed : REFERENCE TO BOOL;
	ShippingHomed : REFERENCE TO BOOL;
	Homed : REFERENCE TO BOOL;
    TimeOut     : LREAL := 120; // Unit : s
	StorageFanucRobot	: FB_FanucRobot_Basic_V2;
	ShippinFanucRobot	: FB_FanucRobot_Basic_V2;
END_VAR
VAR_OUTPUT
	xAborted : BOOL;
	iErrorID : INT;
	ErrorMsg : STRING;
END_VAR
VAR
	StateBehaviour : CBML.ETrigATo;
	uiMachineHomingStep : UINT;
	fbExecuteEdgeDetect :FB_EdgeDetect;
END_VAR

THIS^.IBehaviourModel := StateBehaviour;
StateBehaviour(xExecute := xExecute,
               xAbort := xAbort OR fbExecuteEdgeDetect.xFallingEdge,
               udiTimeOut := LREAL_TO_UDINT( TimeOut*1000000),
               xDone => xDone,
               xBusy => xBusy,
               xError => xError,
               xAborted => xAborted);
			   
//Make sure that C# turns off execute to shut down the service
fbExecuteEdgeDetect(xInput :=xExecute);

iErrorID := StateBehaviour._model.iErrorID;
ErrorMsg := M_GetErrorMsg(xErrorID := iErrorID);

METHOD CleanupAction
VAR_INPUT
    xAbortProposed : BOOL;
    iErrorIDProposed: INT;
END_VAR
VAR_OUTPUT
    xComplete : BOOL := TRUE;
    xAbort: BOOL := xAbortProposed;
 	iErrorID : INT := iErrorIDProposed;
END_VAR
END_METHOD

METHOD CyclicAction
VAR_INPUT
    itfTimingController : CBML.ITimingController;
END_VAR
VAR_OUTPUT
    xComplete : BOOL := TRUE;
    iErrorID : INT := 0;
END_VAR
xComplete := FALSE;
CASE uiMachineHomingStep OF 
	0:
		IF AllocateHome.Homed AND Storagehome.Homed AND Shippinghome.Homed THEN
			Allocatehome.xExecute := TRUE;
			Storagehome.xExecute := TRUE;
			ShippingHome.xExecute := TRUE;
		END_IF
		IF NOT AllocateHome.Homed THEN
			AllocateHome.xExecute := TRUE;
		END_IF
		IF NOT StorageHome.Homed THEN
			StorageHome.xExecute := TRUE;
		END_IF
		IF NOT ShippingHome.Homed THEN
			ShippingHome.xExecute := TRUE;
		END_IF
		uiMachineHomingStep := 100;
	100:
		IF AllocateHome.Homed AND StorageHome.Homed AND ShippingHome.Homed THEN
			uiMachineHomingStep := 200;
		END_IF
	200:
		Homed := TRUE;
		uiMachineHomingStep := 300;
	300:
		xComplete := TRUE;
		// 
END_CASE

//IF StorageFanucRobot.Error THEN
//	iErrorID := 11;
//END_IF
//IF ShippinFanucRobot.Error THEN
//	iErrorID := 12;
//END_IF
END_METHOD

METHOD ExitAction
VAR_INPUT
    xAfterCleanup : BOOL;
    xInCopyCode : BOOL;
END_VAR
END_METHOD

METHOD M_GetErrorMsg : T_MaxString
VAR_INPUT
	xErrorID: INT;
END_VAR

VAR
	
END_VAR
CASE xErrorID OF
    0:
        M_GetErrorMsg := 'No Error';
    1:
        M_GetErrorMsg := 'FB_MachineHoming ErrorID 1: Action time out';
    2:
        M_GetErrorMsg := 'FB_MachineHoming ErrorID 2: Position Data invalid';
    3:
        M_GetErrorMsg := 'FB_MachineHoming ErrorID 3: Index invalid';
    4:
		M_GetErrorMsg := 'FB_MachineHoming ErrorID 4: Axis is not ready';
    5:
        M_GetErrorMsg := 'FB_MachineHoming ErrorID 5: Axis OutRobot X has Error';
    6:
        M_GetErrorMsg := 'FB_MachineHoming ErrorID 6: Axis OutRobot Y has Error';
	7:
		M_GetErrorMsg := 'FB_MachineHoming ErrorID 7: Axis Allocate_X has error';
	8:
		M_GetErrorMsg := 'FB_MachineHoming ErrorID 8: Axis Allocate_Y has error';
	9:
		M_GetErrorMsg := 'FB_MachineHoming ErrorID 9: Axis RoundBelt has error';
	10:
		M_GetErrorMsg := 'FB_MachineHoming ErrorID 10: Axis TurnTable has error';
	11:
		M_GetErrorMsg := StorageFanucRobot.ErrMsg;
	12:
		M_GetErrorMsg := ShippinFanucRobot.ErrMsg;
END_CASE
END_METHOD

METHOD ResetAction
VAR_OUTPUT
    xComplete : BOOL := TRUE;
END_VAR
END_METHOD

METHOD StartAction
VAR_OUTPUT
    xComplete : BOOL := TRUE;
	iErrorID : INT := 0;
END_VAR
xComplete := FALSE;
Homed := FALSE;
uiMachineHomingStep := 0;

//IF StorageFanucRobot.Error THEN
//	iErrorID := 11;
//END_IF
//IF ShippinFanucRobot.Error THEN
//	iErrorID := 12;
//END_IF

xComplete := TRUE;
END_METHOD

END_FUNCTION_BLOCK

// ---- Library/99_Utilities/FB_CylinderManualCtrl.TcPOU
FUNCTION_BLOCK FB_CylinderManualCtrl
VAR_INPUT
	bTrigger	: BOOL;
	Cylinder	: REFERENCE TO  FB_Cylinder; 
	Hold		: BOOL; //Add for holding the cylinder
END_VAR
VAR_OUTPUT
END_VAR
VAR
	rTrig	:R_TRIG;
	fTrig	:F_TRIG;
END_VAR

IF NOT Hold THEN
	rTrig(CLK:=bTrigger);
	fTrig(CLK:=bTrigger);
END_IF

IF rTrig.Q THEN
	Cylinder.M_Extend();
ELSIF fTrig.Q THEN
	Cylinder.M_Retract();
END_IF

END_FUNCTION_BLOCK

// ---- Library/99_Utilities/FB_MotorManualCtrl.TcPOU
{attribute 'hide_all_locals'}
FUNCTION_BLOCK FB_MotorManualCtrl

VAR_INPUT
	bForward	: BOOL;
	bBackward	: BOOL;
	bStop		: BOOL;
	Hold		: BOOL;	//Add for holding the cylinder
	Motor		: REFERENCE TO  FB_Motor; 
END_VAR
VAR_OUTPUT
END_VAR
VAR
	ForWardrTrig	:R_TRIG;
	ForWardfTrig	:F_TRIG;
	
	BackWardrTrig	:R_TRIG;
	BackWardfTrig	:F_TRIG;
	
	
	
END_VAR

IF NOT Hold THEN
	ForWardrTrig(CLK:=bForward);
	ForWardfTrig(CLK:=bForward);
	
	BackWardrTrig(CLK:=bBackward);
	BackWardfTrig(CLK:=bBackward);
END_IF

IF ForWardrTrig.Q AND NOT bBackward AND NOT bStop THEN
	Motor.M_MoveForward();	
END_IF

IF BackWardrTrig.q AND NOT bForward AND NOT bStop THEN
	Motor.M_MoveBackward();
END_IF

IF bStop OR ForWardfTrig.Q OR BackWardfTrig.Q THEN
	Motor.M_MotorStop();
END_IF

END_FUNCTION_BLOCK

// ---- Library/10_Machine/13_ErrorHandling/FB_ErrorHandler_V2.TcPOU
FUNCTION_BLOCK FB_ErrorHandler_V2 EXTENDS FB_ActionBasic
VAR_INPUT
    AlarmList : REFERENCE TO ARRAY[1..Tc3_PackML_V2.MaxAlarms] OF ST_Alarm; // 輸入的錯誤信號矩陣
    HMI_AlarmMonitorList : REFERENCE TO ARRAY[0..999] OF ST_Alarm_Tmax;     // 輸出的錯誤信號矩陣
    AlarmHistory : REFERENCE TO ARRAY[1..Tc3_PackML_V2.MaxHistoryAlarms] OF ST_Alarm;
    MaxRecords : INT := 1000;      // 最大記錄數量
    Reset : BOOL;                  // RESET按鈕
    ResetAllAlarms : BOOL;         // 重置所有錯誤
    EnableLogging : BOOL := TRUE;  // 啟動錯誤紀錄
    ResetDelayTime : TIME := T#1.5S; // RESET後延遲確認時間
END_VAR
VAR_OUTPUT
    ActiveAlarmCount : INT;    // 活動錯誤數量
    TotalRecords : INT;        // 總記錄數量
    SystemStatus : STRING(50); // 系統狀態
    CurrentSeverityLevel : DINT; // 當前最高嚴重程度 (1-7, 7最嚴重)
	IsResetting : BOOL;       // 正在執行RESET程序
END_VAR
VAR
    // 內部變量
    i : INT;
    j : INT;
	k : INT;
    CurrentTime : DATE_AND_TIME;
    LastTriggerState : ARRAY[1..200] OF BOOL; // 上次Trigger狀態記錄
    RisingEdge : ARRAY[1..200] OF BOOL;       // 上升沿檢測
    FallingEdge : ARRAY[1..200] OF BOOL;      // 下降沿檢測
    RecordIndex : INT := 0;                   // 記錄索引
    HistoryIndex : INT := 1;                  // 歷史記錄索引
    // 邊沿檢測功能塊
    R_TRIG_Array : ARRAY[1..200] OF R_TRIG;
    F_TRIG_Array : ARRAY[1..200] OF F_TRIG;

    // 時間相關
    fbLocalSystemTime : FB_LocalSystemTime := (bEnable := TRUE, dwCycle := 30);
	fbNtTime : GETSYSTEMTIME;
	SystemTimeStruct : TIMESTRUCT;
	_PackMLTime : ARRAY[0..6] OF DINT;
    // 排序用的臨時變數
    TempAlarm : ST_Alarm_Tmax;
    bNeedSort : BOOL;
    TempHistoryAlarm : ST_Alarm; // 歷史記錄排序用
    bNeedHistorySort : BOOL;     // 歷史記錄需要排序
    // 時間比較用的變數
    TimeCompareResult : INT;        // -1:j較舊, 0:相等, 1:j較新
    HistoryTimeCompareResult : INT; // 歷史記錄時間比較結果
    TimeIndex : INT;
	 // 確認機制用的變數
    R_TRIG_Reset : R_TRIG;       // RESET按鈕邊沿檢測
    R_TRIG_Start : R_TRIG;       // START按鈕邊沿檢測
    AllAlarmsCleared : BOOL;     // 所有錯誤都已清除
	// 延遲確認機制
    TON_ResetDelay : TON;        // RESET延遲確認計時器
    ResetInProgress : BOOL;      // RESET程序進行中
    ResetPendingList : ARRAY[0..999] OF BOOL; // 待確認清除的錯誤列表
	defaultST_Alarm_Tmax : ST_Alarm_Tmax;
END_VAR


// 主要執行程序
fbLocalSystemTime();
_PackMLTime := TIMESTRUCT_TO_PackMLTime(fbLocalSystemTime.systemTime);

ActiveAlarmCount := 0;

// RESET按鈕邊沿檢測
R_TRIG_Reset(CLK := Reset);

// RESET延遲確認計時器
TON_ResetDelay(IN := ResetInProgress, PT := ResetDelayTime);
IsResetting := ResetInProgress;

// RESET按鈕延遲確認機制
IF R_TRIG_Reset.Q THEN
    // 啟動RESET程序
    ResetInProgress := TRUE;
    
    // 標記所有當前錯誤為待確認狀態
    FOR i := 0 TO TotalRecords - 1 DO
        ResetPendingList[i] := (HMI_AlarmMonitorList[i].ID <> 0);
		//HMI_AlarmMonitorList[i] :=defaultST_Alarm_Tmax; // remove error anyway
    END_FOR;
END_IF;

// RESET延遲時間到達，開始確認錯誤狀態
IF TON_ResetDelay.Q AND ResetInProgress THEN
    ResetInProgress := FALSE;
    
    // 延遲確認：檢查每個標記的錯誤是否真正清除
    FOR i := 0 TO TotalRecords - 1 DO
        IF ResetPendingList[i] AND HMI_AlarmMonitorList[i].ID <> 0 THEN
            // 檢查該錯誤在AlarmList中的對應項目是否已經清除
            FOR j := 1 TO Tc3_PackML_V2.MaxAlarms DO
                IF AlarmList[j].ID = UDINT_TO_DINT( HMI_AlarmMonitorList[i].ID) THEN
                    // 找到對應的錯誤源
                    IF NOT AlarmList[j].Trigger THEN
                        // 錯誤已清除，可以移到歷史記錄
                        IF HistoryIndex <= Tc3_PackML_V2.MaxHistoryAlarms THEN
                            // 搬移到AlarmHistory
                            AlarmHistory[HistoryIndex].ID := UDINT_TO_DINT(HMI_AlarmMonitorList[i].ID);
                            AlarmHistory[HistoryIndex].Trigger := FALSE;
                            AlarmHistory[HistoryIndex].Category := HMI_AlarmMonitorList[i].Category;
                            AlarmHistory[HistoryIndex].Value := HMI_AlarmMonitorList[i].Value;
                            AlarmHistory[HistoryIndex].Message := HMI_AlarmMonitorList[i].Message;
                            
                            // 複製發生時間
                            AlarmHistory[HistoryIndex].DateTime := HMI_AlarmMonitorList[i].DateTime;
                            
                            // 記錄清除時間
                            AlarmHistory[HistoryIndex].AckDateTime := _PackMLTime;
                            
                            HistoryIndex := HistoryIndex + 1;
                            IF HistoryIndex > Tc3_PackML_V2.MaxHistoryAlarms THEN
                                HistoryIndex := 1;
                            END_IF;
                        END_IF;
                        
                        // 清空HMI記錄
                        HMI_AlarmMonitorList[i].ID := 0;
                        HMI_AlarmMonitorList[i].Trigger := FALSE;
                        HMI_AlarmMonitorList[i].Category := 0;
                        HMI_AlarmMonitorList[i].Value := 0;
                        HMI_AlarmMonitorList[i].Message := '';
                        HMI_AlarmMonitorList[i].DateTime := DT_TO_PackMLTime(DT#1970-01-01-00:00:00);
                        HMI_AlarmMonitorList[i].ackDateTime := DT_TO_PackMLTime(DT#1970-01-01-00:00:00);
                        
                        bNeedSort := TRUE;
                        bNeedHistorySort := TRUE;
                    END_IF;
                    EXIT; // 找到對應項目，跳出內層迴圈
                END_IF;
            END_FOR;
        END_IF;
        // 清除待確認標記
        ResetPendingList[i] := FALSE;
    END_FOR;
END_IF;

// 邊沿檢測和錯誤處理
FOR i := 1 TO Tc3_PackML_V2.MaxAlarms DO
    // 上升沿檢測 - 錯誤發生
    R_TRIG_Array[i](CLK := AlarmList[i].Trigger);
    RisingEdge[i] := R_TRIG_Array[i].Q;
    
    // 下降沿檢測 - 錯誤清除
    F_TRIG_Array[i](CLK := AlarmList[i].Trigger);
    FallingEdge[i] := F_TRIG_Array[i].Q;
    
    // 處理錯誤發生 (上升沿)
    IF AlarmList[i].Trigger AND EnableLogging THEN
        // 檢查是否已存在相同的活動錯誤
        j := -1;  // 初始化為-1，表示未找到
        FOR k := 0 TO TotalRecords - 1 DO
            IF HMI_AlarmMonitorList[k].ID = DINT_TO_UDINT( AlarmList[i].ID ) AND
                HMI_AlarmMonitorList[k].Trigger THEN
                j := k;  // 找到重複錯誤，記錄位置
                EXIT; // 已存在活動錯誤，跳出
            END_IF;
        END_FOR;
        
        // 如果沒有找到重複的活動錯誤，創建新記錄
        IF j = -1 THEN
            // 尋找空的位置插入新錯誤
            FOR k := 0 TO MaxRecords - 1 DO
                IF HMI_AlarmMonitorList[k].ID = 0 THEN
                    // 找到空位置，插入新錯誤
                    HMI_AlarmMonitorList[k].ID := DINT_TO_UDINT(AlarmList[i].ID);
                    HMI_AlarmMonitorList[k].Trigger := TRUE;
                    HMI_AlarmMonitorList[k].Category := AlarmList[i].Category;
                    HMI_AlarmMonitorList[k].Value := AlarmList[i].Value;
                    HMI_AlarmMonitorList[k].Message := AlarmList[i].Message;
                    
                    // 填入發生時間
                    HMI_AlarmMonitorList[k].DateTime := _PackMLTime;
                    HMI_AlarmMonitorList[k].ackDateTime := DT_TO_PackMLTime(DT#1970-01-01-00:00:00);
                    
                    // 更新記錄統計
                    TotalRecords := TotalRecords + 1;
                    bNeedSort := TRUE;
                    
                    EXIT; // 插入完成，跳出迴圈
                END_IF;
            END_FOR;
        END_IF;
    END_IF;
    
    // 處理錯誤清除 - 修正：移除自動清除邏輯
    // 不再監控下降沿自動清除，只等待RESET按鈕手動清除
    // IF FallingEdge[i] AND EnableLogging THEN
    //     // 此段程式碼已移除，改為只在RESET時處理
    // END_IF;
    
    // 統計活動錯誤數量
    IF AlarmList[i].Trigger THEN
        ActiveAlarmCount := ActiveAlarmCount + 1;
    END_IF;
END_FOR;

// 如果有資料異動，重新排序HMI_AlarmMonitorList
// 保持錯誤記錄不被清除，只排序顯示順序
IF bNeedSort THEN
    // 簡化排序：只按時間排序，不清除任何記錄
    FOR i := 0 TO MaxRecords - 2 DO
        FOR j := 0 TO MaxRecords - 2 - i DO
            // 只有兩個位置都有有效記錄才比較
            IF HMI_AlarmMonitorList[j].ID <> 0 AND HMI_AlarmMonitorList[j+1].ID <> 0 THEN
                
                // 比較發生時間，較新的排在前面
                TimeCompareResult := 0;
                FOR TimeIndex := 0 TO 5 DO
                    IF HMI_AlarmMonitorList[j].DateTime[TimeIndex] < HMI_AlarmMonitorList[j+1].DateTime[TimeIndex] THEN
                        TimeCompareResult := -1; // j較舊
                        EXIT;
                    ELSIF HMI_AlarmMonitorList[j].DateTime[TimeIndex] > HMI_AlarmMonitorList[j+1].DateTime[TimeIndex] THEN
                        TimeCompareResult := 1; // j較新
                        EXIT;
                    END_IF;
                END_FOR;
                
                // 如果j較舊，交換位置（較新的往前）
                IF TimeCompareResult = -1 THEN
                    TempAlarm := HMI_AlarmMonitorList[j];
                    HMI_AlarmMonitorList[j] := HMI_AlarmMonitorList[j+1];
                    HMI_AlarmMonitorList[j+1] := TempAlarm;
                END_IF;
            END_IF;
        END_FOR;
    END_FOR;
    
    // 重新計算TotalRecords（所有有效記錄，不管Trigger狀態）
    TotalRecords := 0;
    FOR i := 0 TO MaxRecords - 1 DO
        IF HMI_AlarmMonitorList[i].ID <> 0 THEN
            TotalRecords := TotalRecords + 1;
        END_IF;
    END_FOR;
    
    bNeedSort := FALSE;
END_IF;

// 如果歷史記錄有新資料，重新排序AlarmHistory (使用PackMLTime比較)
IF bNeedHistorySort THEN
    // 使用泡沫排序法排序歷史記錄 (按DateTime由新到舊)
    FOR i := 1 TO Tc3_PackML_V2.MaxHistoryAlarms - 1 DO
        FOR j := 1 TO Tc3_PackML_V2.MaxHistoryAlarms - i DO
            // 只排序有效的記錄 (ID不為0)
            IF AlarmHistory[j].ID <> 0 AND AlarmHistory[j+1].ID <> 0 THEN
                
                // 比較兩個時間：j vs j+1
                HistoryTimeCompareResult := 0;
                
                // 比較PackMLTime陣列
                FOR TimeIndex := 0 TO 5 DO
                    IF AlarmHistory[j].DateTime[TimeIndex] < AlarmHistory[j+1].DateTime[TimeIndex] THEN
                        HistoryTimeCompareResult := -1; // j較舊
                        EXIT;
                    ELSIF AlarmHistory[j].DateTime[TimeIndex] > AlarmHistory[j+1].DateTime[TimeIndex] THEN
                        HistoryTimeCompareResult := 1; // j較新
                        EXIT;
                    END_IF;
                END_FOR;
                
                // 如果j較舊，則交換位置（讓較新的往前移）
                IF HistoryTimeCompareResult = -1 THEN
                    TempHistoryAlarm := AlarmHistory[j];
                    AlarmHistory[j] := AlarmHistory[j+1];
                    AlarmHistory[j+1] := TempHistoryAlarm;
                END_IF;
            END_IF;
        END_FOR;
    END_FOR;
    
    bNeedHistorySort := FALSE;
END_IF;

// 更新系統狀態和嚴重程度
CurrentSeverityLevel := 0; // 初始化為無錯誤

// 掃描HMI_AlarmMonitorList中活動錯誤的最高嚴重程度
FOR i := 0 TO TotalRecords - 1 DO
    IF HMI_AlarmMonitorList[i].Trigger THEN  // 只計算活動錯誤
        // 找出最高嚴重程度
        IF HMI_AlarmMonitorList[i].Value > CurrentSeverityLevel THEN
            CurrentSeverityLevel := HMI_AlarmMonitorList[i].Value;
        END_IF;
    END_IF;
END_FOR;

// 統計真正的活動錯誤數量（Trigger=TRUE）
ActiveAlarmCount := 0;
FOR i := 0 TO TotalRecords - 1 DO
    IF HMI_AlarmMonitorList[i].Trigger THEN
        ActiveAlarmCount := ActiveAlarmCount + 1;
    END_IF;
END_FOR;

END_FUNCTION_BLOCK

// ---- Library/99_Utilities/FB_SignalTower.TcPOU
FUNCTION_BLOCK FB_SignalTower
VAR_INPUT
    // TRUE: Activates the defined operation
    // FALSE: Aborts/resets the defined operation
    Enable     :BOOL := TRUE;
    LampRed    :REFERENCE TO BOOL;
    LampYellow :REFERENCE TO BOOL;
    LampGreen  :REFERENCE TO BOOL;
    Buzz       :REFERENCE TO BOOL;
	ForceCloseBuzz : BOOL;
	BuzzSwitchOnTime	:LREAL :=3000.0 ; //In Second
END_VAR

VAR_OUTPUT
    // TRUE: Operation is running
    Vaild :BOOL;
    // TRUE: Error condition reached
    Error :BOOL;
    // Error code describing error condition
    ErrorID :DINT;
END_VAR

VAR
    LampRed_Active    :BOOL;         // True :Lamp Red actived
    LampYellow_Active :BOOL;         // True :Lamp Yellow actived
    LampGreen_Active  :BOOL;         // True : Lamp Green actived
    FB_1Hz            :FB_SignalGen; // 1Hz flash signal generator
    FB_2Hz            :FB_SignalGen; // 2Hz flash signal generator
    FB_05Hz           :FB_SignalGen; // 0.5 Hz flash signal generator
    // Signal Tower controller output
    LampSingal :ST_SignalTower;
	BuzzOnTimer			:TON;
	bBuzzBypass			: BOOL;
END_VAR

// Call Signal generator
A_SignalGenerator();

// 
IF Enable THEN
	LampSingal.Lamp_Red 	:= M_LampRed();
	LampSingal.Lamp_Yellow	:= M_LampYellow();
	LampSingal.Lamp_Green 	:= M_LampGreen();
	LampSingal.Buzz			:=M_Buzz(BuzzSwitchOnTime);
ELSE
	LampSingal.Lamp_Red := FALSE;
	LampSingal.Lamp_Yellow := FALSE;
	LampSingal.Lamp_Green := FALSE;
	LampSingal.Buzz := FALSE;
END_IF

LampRed := LampSingal.Lamp_Red;
LampYellow := LampSingal.Lamp_Yellow;
LampGreen := LampSingal.Lamp_Green;
Buzz := LampSingal.Buzz;

IF GVL_ADS.MachineState <> E_MachineState.Error THEN
	bBuzzBypass := FALSE;
ELSIF GVL_ADS.MachineState = E_MachineState.Error AND 
		GVL_ADS.OpPannel_Status.StartBtnStatus THEN 
	bBuzzBypass := TRUE;
END_IF

ACTION A_SignalGenerator:
FB_1Hz(PT := F_FtoPT(Hz := 1));
FB_2Hz(PT := F_FtoPT(Hz := 2));
FB_05Hz(PT := F_FtoPT(Hz := 0.5));
END_ACTION

METHOD M_Buzz : BOOL
VAR_INPUT
	SwitchOnTime : LREAL ;//In second
END_VAR
VAR
	SignalMode: E_SignalTowerLampMode:=E_SignalTowerLampMode.Disable;
	
END_VAR
BuzzOnTimer(PT:= DWORD_TO_TIME(LREAL_TO_DWORD(SwitchOnTime*1000)));

IF ForceCloseBuzz THEN
	SignalMode := E_SignalTowerLampMode.Disable;
ELSE
	IF  GVL_ADS.MachineState = E_MachineState.Error THEN
		BuzzOnTimer.IN :=TRUE;		
		IF NOT bBuzzBypass THEN			// 泰興客戶需要長時間鳴笛時，有手段可以 bypass 鳴笛
			SignalMode := E_SignalTowerLampMode.Flash_2Hz;
		END_IF			
	ELSE   
		BuzzOnTimer.IN :=FALSE;
	END_IF
	
END_IF
// Determine the Lamp mode based on the current SignalTowerMode. 
CASE SignalMode OF
    E_SignalTowerLampMode.Disable: // Lamp off
        M_Buzz := FALSE;
    E_SignalTowerLampMode.AlwaysOn: // Lamp on
        M_Buzz := TRUE AND NOT BuzzOnTimer.Q;
    E_SignalTowerLampMode.Flash_05Hz: // Lamp flash 0.25s on 0.25s off
        M_Buzz := FB_05Hz.Q AND NOT BuzzOnTimer.Q;
    E_SignalTowerLampMode.Flash_1Hz: // Lamp flash 0.5s on 0.5s off	
        M_Buzz := FB_1Hz.Q AND NOT BuzzOnTimer.Q ;
    E_SignalTowerLampMode.Flash_2Hz: // Lamp flash 1s on 1s off
        M_Buzz := FB_2Hz.Q AND ( NOT BuzzOnTimer.Q);
END_CASE
END_METHOD

METHOD M_LampGreen : BOOL
VAR_INPUT
END_VAR
VAR
	SignalMode: E_SignalTowerLampMode:=E_SignalTowerLampMode.Disable;
END_VAR
IF NOT LampRed_Active  THEN
    IF GVL_ADS.MachineState=E_MachineState.Running THEN
        SignalMode := E_SignalTowerLampMode.AlwaysOn;
    ELSE
        SignalMode := E_SignalTowerLampMode.Disable;
    END_IF
ELSIF LampRed_Active  THEN
    SignalMode := E_SignalTowerLampMode.Disable;
END_IF;

// Determine the Lamp mode based on the current SignalTowerMode. 
CASE SignalMode OF
    E_SignalTowerLampMode.Disable: // Lamp off
        M_LampGreen := FALSE;
    E_SignalTowerLampMode.AlwaysOn: // Lamp on
        M_LampGreen := TRUE;
    E_SignalTowerLampMode.Flash_05Hz: // Lamp flash 0.25s on 0.25s off
        M_LampGreen := FB_05Hz.Q;
    E_SignalTowerLampMode.Flash_1Hz: // Lamp flash 0.5s on 0.5s off	
        M_LampGreen := FB_1Hz.Q;
    E_SignalTowerLampMode.Flash_2Hz: // Lamp flash 1s on 1s off
        M_LampGreen := FB_2Hz.Q;
END_CASE

// Lamp effective flag
IF SignalMode = E_SignalTowerLampMode.Disable THEN
    LampGreen_Active := FALSE;
ELSE
    LampGreen_Active := TRUE;
END_IF
END_METHOD

METHOD M_LampRed : BOOL
VAR_INPUT
END_VAR
VAR
	SignalMode: E_SignalTowerLampMode:=E_SignalTowerLampMode.Disable;
END_VAR
// Control SignalMode here
IF GVL_ADS.MachineState=E_MachineState.Error THEN
	SignalMode := E_SignalTowerLampMode.Flash_1Hz;
ELSIF GVL_ADS.MachineState=E_MachineState.StandBy THEN
	SignalMode := E_SignalTowerLampMode.AlwaysOn;	
ELSE
	SignalMode := E_SignalTowerLampMode.Disable;
END_IF
// Determine the Lamp mode based on the current SignalTowerMode. 
CASE SignalMode OF
    E_SignalTowerLampMode.Disable: // Lamp off
        M_LampRed := FALSE;
    E_SignalTowerLampMode.AlwaysOn:// Lamp on
        M_LampRed := TRUE;
    E_SignalTowerLampMode.Flash_05Hz:// Lamp flash 0.25s on 0.25s off
        M_LampRed := FB_05Hz.Q;
    E_SignalTowerLampMode.Flash_1Hz: // Lamp flash 0.5s on 0.5s off
        M_LampRed := FB_1Hz.Q;
    E_SignalTowerLampMode.Flash_2Hz: // Lamp flash 1s on 1s off
        M_LampRed := FB_2Hz.Q;
END_CASE
// Lamp effective flag
IF SignalMode = E_SignalTowerLampMode.Disable THEN
	LampRed_Active := FALSE;
ELSE
	LampRed_Active := TRUE;
END_IF
END_METHOD

METHOD M_LampYellow : BOOL
VAR_INPUT
END_VAR
VAR
	SignalMode: E_SignalTowerLampMode:=E_SignalTowerLampMode.Disable;
END_VAR
// Contorl Signal here
 IF GVL_ADS.MachineState=E_MachineState.NotHomed OR GVL_ADS.MachineState=E_MachineState.Homing THEN
	
		SignalMode := E_SignalTowerLampMode.Flash_2Hz;
	ELSIF GVL_ADS.MachineState=E_MachineState.Homed THEN
		SignalMode := E_SignalTowerLampMode.AlwaysOn;
	ELSE	
		SignalMode := E_SignalTowerLampMode.Disable;
	
END_IF

// Determine the Lamp mode based on the current SignalTowerMode. 
CASE SignalMode OF
    E_SignalTowerLampMode.Disable: // Lamp off
        M_LampYellow := FALSE;
    E_SignalTowerLampMode.AlwaysOn:// Lamp on
        M_LampYellow := TRUE;
    E_SignalTowerLampMode.Flash_05Hz:// Lamp flash 0.25s on 0.25s off
        M_LampYellow := FB_05Hz.Q;
    E_SignalTowerLampMode.Flash_1Hz: // Lamp flash 0.5s on 0.5s off
        M_LampYellow := FB_1Hz.Q;
    E_SignalTowerLampMode.Flash_2Hz: // Lamp flash 1s on 1s off
        M_LampYellow := FB_2Hz.Q;
END_CASE
// Lamp effective flag
IF SignalMode = E_SignalTowerLampMode.Disable THEN
	LampYellow_Active := FALSE;
ELSE
	LampYellow_Active := TRUE;
END_IF
END_METHOD

PROPERTY PUBLIC P_LampGreenState : Bool
GET
P_LampGreenState:=LampSingal.Lamp_Green ;
END_GET
END_PROPERTY

PROPERTY PUBLIC P_LampRedState : Bool
GET
P_LampRedState:=LampSingal.Lamp_Red ;
END_GET
END_PROPERTY

PROPERTY PUBLIC P_LampYellowState : Bool
GET
P_LampYellowState:=LampSingal.Lamp_Yellow ;
END_GET
END_PROPERTY

END_FUNCTION_BLOCK

// ---- Library/10_Machine/12_MachineControl/Service/FB_BuzzCtrl.TcPOU
FUNCTION_BLOCK FB_BuzzCtrl EXTENDS FB_ObjectBase_V2
VAR_INPUT
	Timer	: LREAL;
  (*Execute    :BOOL;   // True : This prog will start.
    Abort      :BOOL;   // True : This prog will be abort.
    Reset      :BOOL;   // True : This prog will be reset.
    ObjectName :STRING; // Set this fb name(About it's action)	*)
END_VAR
VAR_OUTPUT
	Buzz	: BOOL;
	(*Busy    :BOOL;        // True : This prog is running.
    Done    :BOOL;        // True : Command has been executed.
    Aborted :BOOL;        // True : This prog is aborted.
    Error   :BOOL;        // True : This prog has an error.
    ErrorID :UINT;       // Output ErrorID
    Status  :T_MaxString; // Output this prog status by string(255bytes)
	UniqueErrorCode :STRING;	*)
END_VAR
VAR
	BuzzBilnker	: BLINK;
	_Timer		: TIME;
	TON_Timer	: TON;
	
	strStatus	: STRING;
END_VAR

SUPER^.A10_StateControl();
THIS^.A00_BasicUnits();

ACTION A00_BasicUnits:
_Timer := LREAL_TO_TIME(Timer*1000);
TON_Timer(PT := _Timer);
BuzzBilnker( TIMEHIGH := T#0.5S , TIMELOW :=T#0.5S );
END_ACTION

METHOD  M_STATE_ABORTED
VAR_INPUT
END_VAR
END_METHOD

METHOD  M_STATE_ABORTING
VAR_INPUT
END_VAR
END_METHOD

METHOD  M_STATE_DONE
VAR_INPUT
END_VAR
Busy := FALSE;
Done := TRUE;

IF NOT Execute THEN
	eSTATE:=STATE_RESETTING;
END_IF
END_METHOD

METHOD  M_STATE_DORMANT
VAR_INPUT
END_VAR
Busy            := FALSE;
Done            := FALSE;
Aborted         := FALSE;
Error           := FALSE;
ErrorID         := 0;
Status          := '';
_ResetCompleted := FALSE;
_AbortCompleted := FALSE;
_Error          := FALSE;
_Executed       := FALSE;
strStatus :='No Error';
uiExecutingStep :=uiResettingStep :=uiAbortingStep :=0;

IF Execute THEN 
	eState := STATE_EXECUTING;
END_IF
END_METHOD

METHOD  M_STATE_ERROR
VAR_INPUT
END_VAR
END_METHOD

METHOD  M_STATE_EXECUTING
VAR_INPUT
END_VAR
Busy := true;
CASE uiExecutingStep OF 
	0:
			uiExecutingStep := 100;
		
	100:
			TON_Timer.IN 		:= TRUE;
			BuzzBilnker.ENABLE  := TRUE;
			BuzzBilnker(OUT => buzz);
			IF TON_Timer.Q THEN 
				BuzzBilnker.ENABLE := FALSE;
				uiExecutingStep := 9900;
			END_IF
	9900:
			Buzz := BuzzBilnker.OUT AND BuzzBilnker.ENABLE;
			strStatus := 'FB_BuzzCtrl Step 9900: Process done ';
			_Executed := TRUE;
	
END_CASE


IF _Executed THEN 
	eState := STATE_DONE;
END_IF
IF NOT Execute THEN
	eState := STATE_RESETTING;
END_IF
END_METHOD

METHOD  M_STATE_RESETTING
VAR_INPUT
END_VAR
Error :=FALSE;
Busy := FALSE;

TON_Timer.IN		:= FALSE;
BuzzBilnker.ENABLE 	:= FALSE;
_ResetCompleted := TRUE;
Buzz := BuzzBilnker.OUT AND BuzzBilnker.ENABLE;
IF _ResetCompleted THEN
	eState := STATE_DORMANT;
END_IF
END_METHOD

END_FUNCTION_BLOCK

// ---- Library/10_Machine/12_MachineControl/Service/FB_MachineModeSwitch.TcPOU
FUNCTION_BLOCK FB_MachineModeSwitch EXTENDS FB_ObjectBase_V2
VAR_INPUT
	ModeLink 				 : REFERENCE TO ST_Mode;
	MachineCtrl_CurrentMode  : E_UnitMode;
	MachineCtrl_CurrentState : E_PMLState;
	MachineHomed			 : BOOL;
END_VAR
VAR_OUTPUT
	RequestedMode		 : E_UnitMode;
	ModeRequestValid	 : BOOL;
END_VAR
VAR
	eTargetModeCache    : E_MachineMode;

	eActualModeCache    : E_UnitMode;

	strStatus           : STRING;
	_bRetry				: BOOL;
	uiResumeStep		: UDINT;
	
	TON_WaitModeSwitch	: TON;
END_VAR

THIS^.A00_BasicUnits();
SUPER^.A10_StateControl();

IF PackTags[0].Status.UnitModeCurrent = E_UnitMode.Manual THEN
	GVL_ADS.MachineMode.CurrentMode := E_MachineMode.MANUAL;
ELSIF PackTags[0].Status.UnitModeCurrent = E_UnitMode.Auto THEN
	GVL_ADS.MachineMode.CurrentMode := E_MachineMode.AUTO;
END_IF

ACTION A00_BasicUnits:
eTargetModeCache := ModeLink.TargetMode;

eActualModeCache := GVL_Machine.PackTags[0].Status.UnitModeCurrent;

TON_WaitModeSwitch(PT := T#3S);
END_ACTION

METHOD M_CheckCommand : BOOL
VAR_INPUT
END_VAR
IF eTargetModeCache = E_MachineMode.AUTO AND NOT MachineHomed THEN
	strStatus := 'FB_MachineModeSwitch ,Not Homing can not Switch AutoMode not can retry';
	M_CheckCommand:= FALSE;
	RETURN;
END_IF

M_CheckCommand := TRUE;
END_METHOD

METHOD  M_STATE_ABORTED
VAR_INPUT
END_VAR
IF NOT _bRetry THEN
	Busy 	:= FALSE;
	Aborted := TRUE;
	Error 	:= TRUE;
	Status 	:= strStatus;
	uiAbortingStep := 0;
	_AbortCompleted := FALSE;
END_IF

IF reset THEN
	_bRetry := TRUE;
	Error	:= FALSE;
	Aborted	:= FALSE;
END_IF

IF NOT Execute THEN
	eState := STATE_RESETTING;
ELSIF Execute AND _bRetry THEN
	uiExecutingStep := uiResumeStep ;
	status :='';
	eState := STATE_EXECUTING;
END_IF
END_METHOD

METHOD  M_STATE_ABORTING
VAR_INPUT
END_VAR
Busy := FALSE;
Done := FALSE;
Aborted := FALSE;
Error := FALSE;
Status := strStatus;

CASE uiAbortingStep OF
	0:
		ModeRequestValid := FALSE;
		TON_WaitModeSwitch.IN := FALSE;
		_Abort := FALSE;
		_bRetry := FALSE;

		uiAbortingStep := 9999;

	9999:
		_AbortCompleted := TRUE;
END_CASE

IF _AbortCompleted THEN
	eState := STATE_ABORTED;
END_IF
END_METHOD

METHOD  M_STATE_DONE
VAR_INPUT
END_VAR
Busy := FALSE;
Done := TRUE;
Aborted := FALSE;
Error := FALSE;
Status := strStatus;

IF Reset OR NOT Execute THEN
	eState := STATE_RESETTING;
END_IF
END_METHOD

METHOD  M_STATE_DORMANT
VAR_INPUT
END_VAR
Busy := FALSE;
Done := FALSE;
Aborted := FALSE;
Error := FALSE;
Paused := FALSE;
Status := '';
UniqueErrorCode := '';

_Executed := FALSE;
_Error := FALSE;
_Abort := FALSE;
_ResetCompleted := FALSE;
_AbortCompleted := FALSE;
_HoldingCompleted := FALSE;
_HeldCompleted := FALSE;
_UnholdCompleted := FALSE;

uiExecutingStep := 0;
uiResettingStep := 0;
uiAbortingStep 	:= 0;
uiHoldingStep 	:= 0;
uiHeldStep 		:= 0;
uiUnholdStep 	:= 0;
uiResumeStep 	:= 0;

_bRetry := FALSE;
TON_WaitModeSwitch.IN := FALSE;
ModeRequestValid := FALSE;

strStatus := 'Machine mode switch idle';
Status := strStatus;

IF Execute THEN
	eState := STATE_EXECUTING;
END_IF
END_METHOD

METHOD  M_STATE_ERROR
VAR_INPUT
END_VAR
Busy := FALSE;
Error := TRUE;
Status := strStatus;
ModeRequestValid := FALSE;

IF NOT Execute THEN
	eState := STATE_RESETTING;
END_IF
END_METHOD

METHOD  M_STATE_EXECUTING
VAR_INPUT
END_VAR

VAR
	esle: INT;
END_VAR
Busy := TRUE;
Done := FALSE;
Aborted := FALSE;
Error := FALSE;

CASE uiExecutingStep OF
	0:
		IF M_CheckCommand() THEN
			uiExecutingStep := 100;
		ELSE
			_Error := TRUE;
		END_IF

	100:
		CASE eTargetModeCache OF
			E_MachineMode.MANUAL:
				TON_WaitModeSwitch.IN 	:= TRUE;
				RequestedMode 			:= E_UnitMode.Manual;
				ModeRequestValid 		:= TRUE;
				IF eActualModeCache = E_UnitMode.Manual THEN
					uiExecutingStep := 200;
				END_IF
				IF TON_WaitModeSwitch.Q THEN
					strStatus := 'FB_MachineModeSwitch ,Switch ManualMode Timeout';
					_Abort := TRUE;
				END_IF
				IF MachineCtrl_CurrentMode = E_UnitMode.Auto AND 
					MachineCtrl_CurrentState = E_PMLState.ePMLState_Suspended  THEN
					uiResumeStep := 100;
					strStatus 	 := 'FB_MachineModeSwitch ,MachineMode stuck in AutoMode Suspended , cat retry';
					_Abort    	 := TRUE;
				END_IF  

			E_MachineMode.AUTO:
				TON_WaitModeSwitch.IN 	:= TRUE;
				RequestedMode 			:= E_UnitMode.Auto;
				ModeRequestValid 		:= TRUE;
				IF eActualModeCache = E_UnitMode.Auto THEN
					uiExecutingStep := 200;
				END_IF
				IF TON_WaitModeSwitch.Q THEN
					strStatus := 'FB_MachineModeSwitch ,Switch AutoMode Timeout';
					_Abort := TRUE;
				END_IF
		ELSE
			ModeRequestValid := FALSE;
			strStatus := 'FB_MachineModeSwitch ,TargetMode is invalid for verification';
			_Error := TRUE;
		END_CASE

	200:
		ModeLink.CurrentMode := eTargetModeCache;
		
		strStatus := 'Machine mode switch verify complete';
		_Executed := TRUE;
END_CASE

